# B&R Automation Studio project 305841_E00002_0
Automation Studio 4.10.3.60 SP; technology packages: mapp 5.16.1, mappCockpit 5.16.0, mappControl 5.16.0, mappMotion 5.16.2, mappSafety 5.16.0, mappView 5.16.1

## Configuration EchCm_AM

CPU X20CP3586, AutomationRuntime B4.92, Build 6.3.0, Safety 0.0, Vc V4.72.5

### Task classes (Cpu.sw)
```
Cyclic#2 (cycle 6400 us, tolerance 6400 us):
  ProdCycle <- PlcLogic.ProdCycle.prg
  Annunc <- PlcLogic.Annunc.prg
Cyclic#3 (cycle 12000 us, tolerance 12000 us):
  Pendant <- PlcLogic.Pendant.prg
  ProcInputs <- PlcLogic.ProcInputs.prg
  axSpinSM <- PlcLogic.axSpindle.axSpindleSM.prg
  axOutESM <- PlcLogic.axOutE.axOutESM.prg
  axInESM <- PlcLogic.axInE.axInESM.prg
  axZSM <- PlcLogic.axZ.axZSM.prg
  axHwSM <- PlcLogic.axHandwheel.axHwSM.prg
  axCfVfdSM <- PlcLogic.axCfVfd.axCfVfdSM.prg
Cyclic#4 (cycle 48000 us, tolerance 48000 us):
  AxEnable <- PlcLogic.AxEnable.prg
  CuttingFlu <- PlcLogic.CuttingFluidVFD.prg
  OmSafeDev <- PlcLogic.OmSafeDev.prg
  CrCamTbl <- PlcLogic.CutProfile.CutProfileCam.prg
  CutProfile <- PlcLogic.CutProfile.PartCfgCalcs.prg
DataObjects: McAcpSys
NcDataObjects: axSpindleP <- PlcLogic.axSpindle.axSpindleParamTable.dob, axOutEPara <- PlcLogic.axOutE.axOutEParamTable.dob, axInEParam <- PlcLogic.axInE.axInEParamTable.dob, axZParamTa <- PlcLogic.axZ.axZParamTable.dob, Cam1P <- PlcLogic.axInE.Cam1P.dob, Cam1P_Fp <- PlcLogic.axInE.Cam1P_Fp.dob, Cam2P <- PlcLogic.axInE.Cam2P.dob, Cam2P_Fp <- PlcLogic.axInE.Cam2P_Fp.dob, Cam3P <- PlcLogic.axInE.Cam3P.dob, Cam3P_Fp <- PlcLogic.axInE.Cam3P_Fp.dob, Cam4P <- PlcLogic.axInE.Cam4P.dob, Cam4P_Fp <- PlcLogic.axInE.Cam4P_Fp.dob, Cam5P <- PlcLogic.axInE.Cam5P.dob, Cam5P_Fp <- PlcLogic.axInE.Cam5P_Fp.dob, Cam6P <- PlcLogic.axInE.Cam6P.dob, Cam6P_Fp <- PlcLogic.axInE.Cam6P_Fp.dob, McDriveLog
Binaries: udbdef, mvLoader, arflatprv, TCData, FWRules, arcoal, arsvcreg, McAcpSim, McProfGen, McAcpDrv, mCoWebSc, TCLang, OpcUaSrv, DataObject, Settings, iomap, asfw, axCfgZ, Role, ashwac, sysconf, arconfig, ashwd, Config, axCfgInE, axCfgSpin, asiol1, axCfgOutE, Anonymous, User, cockpit1, TC, vAxHwCfg, vAxHw, axCfgCfPmp, CamFeature, camlist1, mappConfig, angleLu, depthLu, vAxHwLin, vAxHwRot, wgRecipe, cmRecipe, HwLinCfg, Config_5, HwRotCfg, Config_3
Libraries: sys_lib, runtime, brsystem, GAProcIO, standard, McBase, SfDomain, MpAxis, McAxis, MpBase, MpRecipe, McAcpAx, GAMpMotion, McPureVAx, astime, AsBrStr, GAConvert, MpAlarmX, AsBrMath, GAMath, CoTrace, AsZip, FileIO, McDS402Ax, MTLookUp, astcp, asieccon, asiodiag, asepl, SfDomDrv, asusb, SfDomVis, aruser, arssl, powerlnk, MpSfDomMgr, dataobj, asioacc, GAMotor, MTFilter, MTBasics, MTTypes
```

### Hardware
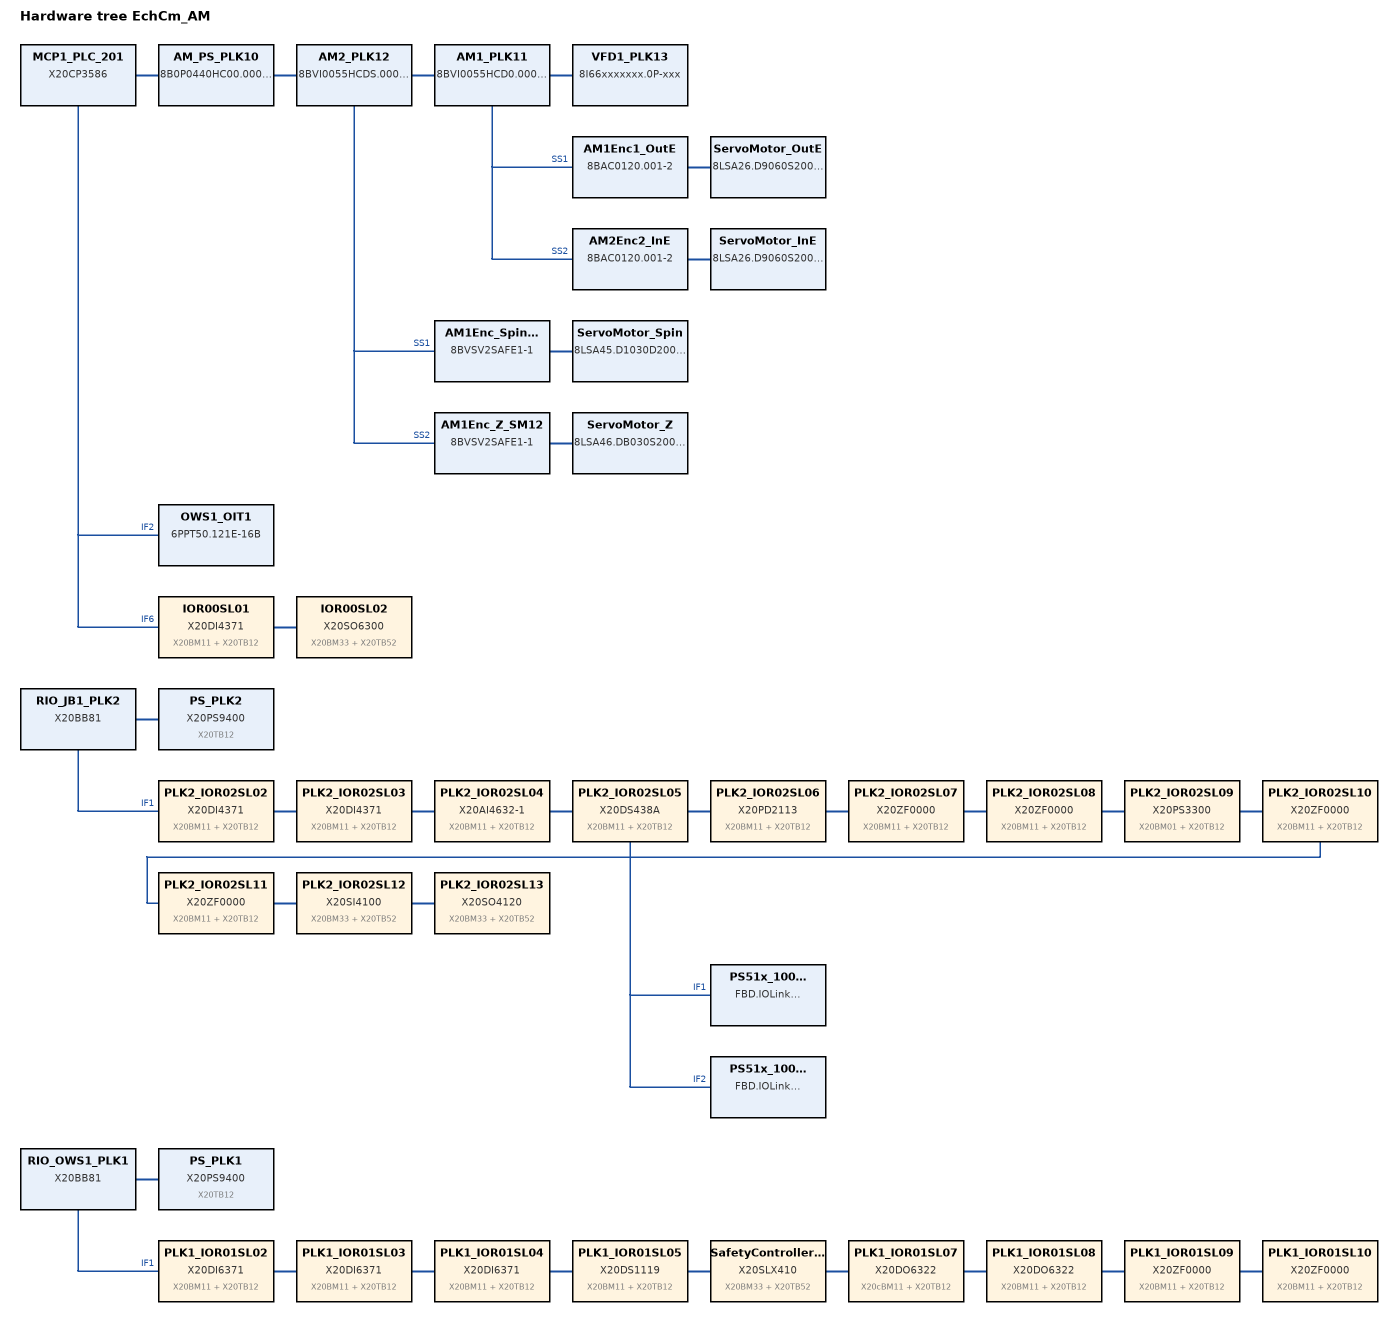
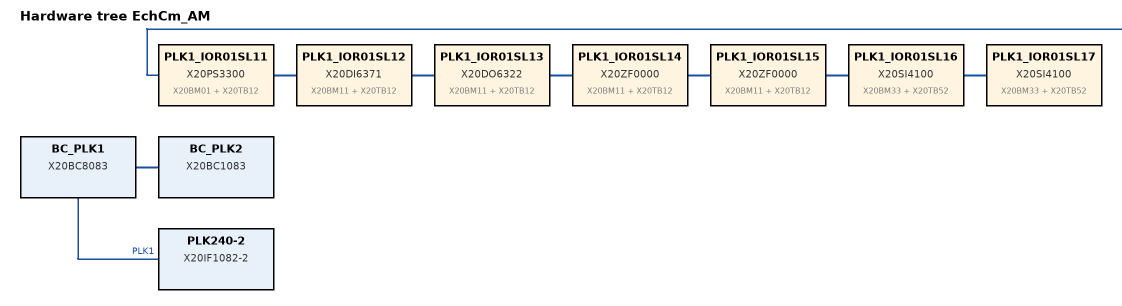
```
AM1Enc1_OutE : 8BAC0120.001-2 v2.2.0.0  [SS -> AM1_PLK11.SS1]
  PlugInType = Encoder
  McAcoposTypeID = AcoposMultiPlugInConfig
AM1Enc_Spin_SM11 : 8BVSV2SAFE1-1 v2.2.0.0  [SS -> AM2_PLK12.SS1]
  SafeModuleID = 11
  PlugInType = Encoder
  McAcoposTypeID = AcoposMultiPlugInConfig
AM1Enc_Z_SM12 : 8BVSV2SAFE1-1 v2.2.0.0  [SS -> AM2_PLK12.SS2]
  SafeModuleID = 12
  PlugInType = Encoder
  McAcoposTypeID = AcoposMultiPlugInConfig
AM1_PLK11 : 8BVI0055HCD0.000-1 v2.3.0.1  [PLK1 -> AM2_PLK12.PLK2 (NodeNumber=11) [Cable Type=PowerlinkCable, Length=10, Version=1.0.0.3]; PLK2 -> VFD1_PLK13.PLK1 (NodeNumber=11) [Cable Type=PowerlinkCable, Length=10, Version=1.0.0.3]; MT2 -> ServoMotor_InE.MT]
  DriveConfiguration/Module:
    McAcoposTypeID = AcoposP3SConfig
    ActivateACOPOSSimulationOnPLC = 0
  DriveConfiguration/Module/PowerSupply:
    PowerSupplyModuleReference = AM_PS
  DriveConfiguration/Channel[1]/RealAxis:
    AxisReference = gAxOutE
    MechanicalElementsIsInvisible = 0
  DriveConfiguration/Channel[1]/RealAxis/MechanicalElements/Gearbox:
    InputIsReadOnly = 0
    Input = 25
    OutputIsReadOnly = 0
    Output = 1
  DriveConfiguration/Channel[1]/RealAxis/MechanicalElements/RotaryToLinearTransformation:
    ReferenceDistanceIsReadOnly = 0
    ReferenceDistance = 360.0
  DriveConfiguration/Channel[1]/RealAxis/Controller:
    ModeIsReadOnly = 0
    Mode = PositionController
  DriveConfiguration/Channel[1]/RealAxis/Controller/Mode/Position:
    ProportionalGain = 462
    IntegrationTime = 0.1
    PredictionTime = 0.0004
    TotalDelayTime = 0.0004
  DriveConfiguration/Channel[1]/RealAxis/Controller/Mode/Speed:
    ProportionalGainIsReadOnly = 0
    ProportionalGain = 0.35
    IntegrationTimeIsReadOnly = 0
    IntegrationTime = 0.0
    FilterTimeIsReadOnly = 0
    FilterTime = 0.0
  DriveConfiguration/Channel[1]/RealAxis/Controller/Mode/LoopFilters:
    LoopFilterXIsReadOnly = 0
    LoopFilter1 = NotUsed
    LoopFilter2 = NotUsed
    LoopFilter3 = NotUsed
  DriveConfiguration/Channel[1]/RealAxis/Homing:
    ModeIsReadOnly = 0
    Mode = RestorePosition
    RestorePositionVariable = ::gr_AxOutERestorePos
  DriveConfiguration/Channel[1]/RealAxis/StopReaction:
    QuickstopIsReadOnly = 0
    Quickstop = DecelerationLimit
    DriveErrorIsReadOnly = 0
    DriveError = DecelerationLimit
  DriveConfiguration/Channel[1]/RealAxis/MovementErrorLimits:
    PositionError = 1.0
    VelocityErrorMonitoring = Automatic1
  DriveConfiguration/Channel[1]/RealAxis:
    JerkFilterIsReadOnly = 0
    JerkFilter = NotUsed
  DriveConfiguration/Channel[1]/RealAxis/DigitalInputs/HomingSwitch:
    SourceIsReadOnly = 0
    Source = NotUsed
    Level = High
  DriveConfiguration/Channel[1]/RealAxis/DigitalInputs/PositiveLimitSwitch:
    SourceIsReadOnly = 0
    Source = NotUsed
    Level = High
  DriveConfiguration/Channel[1]/RealAxis/DigitalInputs/NegativeLimitSwitch:
    SourceIsReadOnly = 0
    Source = NotUsed
    Level = High
  DriveConfiguration/Channel[1]/RealAxis/DigitalInputs/Trigger1:
    Source = X2Trigger1
    Level = High
  DriveConfiguration/Channel[1]/RealAxis/DigitalInputs/Trigger2:
    Source = X2Trigger2
    Level = High
  DriveConfiguration/Channel[1]/RealAxis/DigitalInputs/Quickstop:
    Input = NotUsed
  DriveConfiguration/Channel[1]/RealAxis/Simulation:
    SimulationModeOnPLC = SetValueGeneration
    SimulationModeOnACOPOS = NotUsed
  DriveConfiguration/Channel[1]:
    ExternalEncoderAxis = NotUsed
  DriveConfiguration/Channel[2]/RealAxis:
    AxisReference = gAxInE
    MechanicalElementsIsInvisible = 0
  DriveConfiguration/Channel[2]/RealAxis/MechanicalElements/Gearbox:
    InputIsReadOnly = 0
    Input = 25
    OutputIsReadOnly = 0
    Output = 1
  DriveConfiguration/Channel[2]/RealAxis/MechanicalElements/RotaryToLinearTransformation:
    ReferenceDistanceIsReadOnly = 0
    ReferenceDistance = 360.0
  DriveConfiguration/Channel[2]/RealAxis/Controller:
    ModeIsReadOnly = 0
    Mode = PositionController
  DriveConfiguration/Channel[2]/RealAxis/Controller/Mode/Position:
    ProportionalGain = 451.5
    IntegrationTime = 0.1
    PredictionTime = 0.0004
    TotalDelayTime = 0.0004
  DriveConfiguration/Channel[2]/RealAxis/Controller/Mode/Speed:
    ProportionalGainIsReadOnly = 0
    ProportionalGain = 0.325
    IntegrationTimeIsReadOnly = 0
    IntegrationTime = 0.0
    FilterTimeIsReadOnly = 0
    FilterTime = 0.0
  DriveConfiguration/Channel[2]/RealAxis/Controller/Mode/LoopFilters:
    LoopFilterXIsReadOnly = 0
    LoopFilter1 = NotUsed
    LoopFilter2 = NotUsed
    LoopFilter3 = NotUsed
  DriveConfiguration/Channel[2]/RealAxis/Homing:
    ModeIsReadOnly = 0
    Mode = RestorePosition
    RestorePositionVariable = ::gr_AxInERestorePos
  DriveConfiguration/Channel[2]/RealAxis/StopReaction:
    QuickstopIsReadOnly = 0
    Quickstop = DecelerationLimit
    DriveErrorIsReadOnly = 0
    DriveError = DecelerationLimit
  DriveConfiguration/Channel[2]/RealAxis/MovementErrorLimits:
    PositionError = 0.9
    VelocityErrorMonitoring = Automatic1
  DriveConfiguration/Channel[2]/RealAxis:
    JerkFilterIsReadOnly = 0
    JerkFilter = NotUsed
  DriveConfiguration/Channel[2]/RealAxis/DigitalInputs/HomingSwitch:
    SourceIsReadOnly = 0
    Source = NotUsed
    Level = High
  DriveConfiguration/Channel[2]/RealAxis/DigitalInputs/PositiveLimitSwitch:
    SourceIsReadOnly = 0
    Source = NotUsed
    Level = Low
  DriveConfiguration/Channel[2]/RealAxis/DigitalInputs/NegativeLimitSwitch:
    SourceIsReadOnly = 0
    Source = NotUsed
    Level = Low
  DriveConfiguration/Channel[2]/RealAxis/DigitalInputs/Trigger1:
    Source = X2Trigger1
    Level = High
  DriveConfiguration/Channel[2]/RealAxis/DigitalInputs/Trigger2:
    Source = X2Trigger2
    Level = High
  DriveConfiguration/Channel[2]/RealAxis/DigitalInputs/Quickstop:
    Input = NotUsed
  DriveConfiguration/Channel[2]/RealAxis/Simulation:
    SimulationModeOnPLC = SetValueGeneration
    SimulationModeOnACOPOS = NotUsed
  DriveConfiguration/Channel[2]/RealAxis/AxisFeatures:
    FeatureRef[1] = 
  DriveConfiguration/Channel[2]:
    ExternalEncoderAxis = NotUsed
  DriveConfiguration/Channel[2]/ChannelFeatures:
    FeatureRef[1] = Feature_CamList
AM2Enc2_InE : 8BAC0120.001-2 v2.2.0.0  [SS -> AM1_PLK11.SS2]
  PlugInType = Encoder
  McAcoposTypeID = AcoposMultiPlugInConfig
AM2_PLK12 : 8BVI0055HCDS.000-1 v2.3.0.1  [PLK1 -> AM_PS_PLK10.PLK2 (NodeNumber=12) [Cable Type=PowerlinkCable, Length=10, Version=1.0.0.3]; PLK2 -> AM1_PLK11.PLK1 (NodeNumber=12) [Cable Type=PowerlinkCable, Length=10, Version=1.0.0.3]; MT2 -> ServoMotor_Z.MT]
  DriveConfiguration/Module:
    McAcoposTypeID = AcoposMultiDConfig
    ActivateACOPOSSimulationOnPLC = 0
  DriveConfiguration/Module/PowerSupply:
    PowerSupplyModuleReference = AM_PS
  DriveConfiguration/Channel[1]/RealAxis:
    AxisReference = gAxSpin
    MechanicalElementsIsInvisible = 0
  DriveConfiguration/Channel[1]/RealAxis/MechanicalElements/Gearbox:
    InputIsReadOnly = 0
    Input = 1
    OutputIsReadOnly = 0
    Output = 1
  DriveConfiguration/Channel[1]/RealAxis/MechanicalElements/RotaryToLinearTransformation:
    ReferenceDistanceIsReadOnly = 0
    ReferenceDistance = 1
  DriveConfiguration/Channel[1]/RealAxis/Controller:
    ModeIsReadOnly = 0
    Mode = PositionControllerWithTorqueFeedForward
  DriveConfiguration/Channel[1]/RealAxis/Controller/Mode/Position:
    ProportionalGainIsReadOnly = 0
    ProportionalGain = 200
    IntegrationTimeIsReadOnly = 0
    IntegrationTime = 0.0
    TotalDelayTime = 0.0004
  DriveConfiguration/Channel[1]/RealAxis/Controller/Mode/Speed:
    ProportionalGainIsReadOnly = 0
    ProportionalGain = 0.25
    IntegrationTimeIsReadOnly = 0
    IntegrationTime = 0
    FilterTimeIsReadOnly = 0
    FilterTime = 0
  DriveConfiguration/Channel[1]/RealAxis/Controller/Mode:
    FeedForwardIsReadOnly = 0
    FeedForward = Standard
  DriveConfiguration/Channel[1]/RealAxis/Controller/Mode/FeedForward:
    TorqueLoad = 0.0
    TorquePositive = 0.3405416
    TorqueNegative = 0.3405416
    SpeedTorqueFactor = 0.00008983436
    Inertia = 0.00009823628
    AccelerationFilterTime = 0.0
  DriveConfiguration/Channel[1]/RealAxis/Controller/Mode/LoopFilters:
    LoopFilterXIsReadOnly = 0
    LoopFilter1 = NotUsed
    LoopFilter2 = NotUsed
    LoopFilter3 = NotUsed
  DriveConfiguration/Channel[1]/RealAxis/Homing:
    ModeIsReadOnly = 0
    Mode = RestorePosition
    RestorePositionVariable = ::gr_AxSpinRestorePos
  DriveConfiguration/Channel[1]/RealAxis/StopReaction:
    QuickstopIsReadOnly = 0
    Quickstop = DecelerationLimit
    DriveErrorIsReadOnly = 0
    DriveError = DecelerationLimit
  DriveConfiguration/Channel[1]/RealAxis/MovementErrorLimits:
    PositionError = 2
    VelocityErrorMonitoring = Automatic1
  DriveConfiguration/Channel[1]/RealAxis:
    JerkFilterIsReadOnly = 0
    JerkFilter = NotUsed
  DriveConfiguration/Channel[1]/RealAxis/DigitalInputs/HomingSwitch:
    SourceIsReadOnly = 0
    Source = NotUsed
    Level = High
  DriveConfiguration/Channel[1]/RealAxis/DigitalInputs/PositiveLimitSwitch:
    SourceIsReadOnly = 0
    Source = NotUsed
    Level = High
  DriveConfiguration/Channel[1]/RealAxis/DigitalInputs/NegativeLimitSwitch:
    SourceIsReadOnly = 0
    Source = NotUsed
    Level = High
  DriveConfiguration/Channel[1]/RealAxis/DigitalInputs/Trigger1:
    Source = X2Trigger1
    Level = High
  DriveConfiguration/Channel[1]/RealAxis/DigitalInputs/Trigger2:
    Source = X2Trigger2
    Level = High
  DriveConfiguration/Channel[1]/RealAxis/DigitalInputs/Quickstop:
    Input = NotUsed
  DriveConfiguration/Channel[1]/RealAxis/Simulation:
    SimulationModeOnPLC = SetValueGeneration
    SimulationModeOnACOPOS = NotUsed
  DriveConfiguration/Channel[1]:
    ExternalEncoderAxis = NotUsed
  DriveConfiguration/Channel[2]/RealAxis:
    AxisReference = gAxZ
    MechanicalElementsIsInvisible = 0
  DriveConfiguration/Channel[2]/RealAxis/MechanicalElements/Gearbox:
    InputIsReadOnly = 0
    Input = 1
    OutputIsReadOnly = 0
    Output = 1
  DriveConfiguration/Channel[2]/RealAxis/MechanicalElements/RotaryToLinearTransformation:
    ReferenceDistanceIsReadOnly = 0
    ReferenceDistance = 5.00
  DriveConfiguration/Channel[2]/RealAxis/Controller:
    ModeIsReadOnly = 0
    Mode = PositionController
  DriveConfiguration/Channel[2]/RealAxis/Controller/Mode/Position:
    ProportionalGain = 551
    IntegrationTime = 0.0
    PredictionTime = 0.0004
    TotalDelayTime = 0.0004
  DriveConfiguration/Channel[2]/RealAxis/Controller/Mode/Speed:
    ProportionalGainIsReadOnly = 0
    ProportionalGain = 1.0
    IntegrationTimeIsReadOnly = 0
    IntegrationTime = 0.0
    FilterTimeIsReadOnly = 0
    FilterTime = 0.0
  DriveConfiguration/Channel[2]/RealAxis/Controller/Mode/LoopFilters:
    LoopFilterXIsReadOnly = 0
    LoopFilter1 = NotUsed
    LoopFilter2 = NotUsed
    LoopFilter3 = NotUsed
  DriveConfiguration/Channel[2]/RealAxis/Homing:
    ModeIsReadOnly = 0
    Mode = RestorePosition
    RestorePositionVariable = ::gr_AxZRestorePos
  DriveConfiguration/Channel[2]/RealAxis/StopReaction:
    QuickstopIsReadOnly = 0
    Quickstop = DecelerationLimit
    DriveErrorIsReadOnly = 0
    DriveError = DecelerationLimit
  DriveConfiguration/Channel[2]/RealAxis/MovementErrorLimits:
    PositionError = 1.0
    VelocityErrorMonitoring = Automatic1
  DriveConfiguration/Channel[2]/RealAxis:
    JerkFilterIsReadOnly = 0
    JerkFilter = NotUsed
  DriveConfiguration/Channel[2]/RealAxis/DigitalInputs/HomingSwitch:
    SourceIsReadOnly = 0
    Source = NotUsed
    Level = High
  DriveConfiguration/Channel[2]/RealAxis/DigitalInputs/PositiveLimitSwitch:
    SourceIsReadOnly = 0
    Source = X2Trigger1
    Level = Low
  DriveConfiguration/Channel[2]/RealAxis/DigitalInputs/NegativeLimitSwitch:
    SourceIsReadOnly = 0
    Source = X2Trigger2
    Level = Low
  DriveConfiguration/Channel[2]/RealAxis/DigitalInputs/Trigger1:
    Source = X2Trigger1
    Level = High
  DriveConfiguration/Channel[2]/RealAxis/DigitalInputs/Trigger2:
    Source = X2Trigger2
    Level = High
  DriveConfiguration/Channel[2]/RealAxis/DigitalInputs/Quickstop:
    Input = NotUsed
  DriveConfiguration/Channel[2]/RealAxis/Simulation:
    SimulationModeOnPLC = SetValueGeneration
    SimulationModeOnACOPOS = NotUsed
  DriveConfiguration/Channel[2]/RealAxis/AxisFeatures:
    FeatureRef[1] = 
  DriveConfiguration/Channel[2]:
    ExternalEncoderAxis = NotUsed
AM_PS_PLK10 : 8B0P0440HC00.000-1 v2.3.0.1  [PLK1 -> MCP1_PLC_201.IF3 (NodeNumber=10) [Cable Type=PowerlinkCable, Length=10, Version=1.0.0.3]; PLK2 -> AM2_PLK12.PLK1 (NodeNumber=10) [Cable Type=PowerlinkCable, Length=10, Version=1.0.0.3]]
  DriveConfiguration/Module:
    McAcoposTypeID = AcoposMultiPSMpConfig
    ActivateACOPOSSimulationOnPLC = 0
  DriveConfiguration/Channel[1]/PowerSection:
    AxisReference = AM_PS
BC_PLK1 : X20BC8083 v2.14.0.0  [PLK1 -> PLK240-2.PLK2 (NodeNumber=1) [Cable Type=PowerlinkCable, Length=10, Version=1.0.0.3]; PLK2 -> BC_PLK2.PLK1 (NodeNumber=1) [Cable Type=PowerlinkCable, Length=10, Version=1.0.0.3]; SL -> RIO_OWS1_PLK1.SL1]
BC_PLK2 : X20BC1083 v2.14.0.0  [PLK1 -> BC_PLK1.PLK2 (NodeNumber=2) [Cable Type=PowerlinkCable, Length=10, Version=1.0.0.3]; SL -> RIO_JB1_PLK2.SL1]
IOR00SL01 : X20DI4371 v1.2.0.0  [SS1 -> X20TB12.SS; SL -> X20BM11.SL1]
IOR00SL02 : X20SO6300 v2.3.0.0  [SS1 -> X20TB52d.SS; SL -> X20BM33d.SL1]
  DigitalOutput01 = viaSafeLOGIC
  DigitalOutput02 = viaSafeLOGIC
  DigitalOutput03 = viaSafeLOGIC
  DigitalOutput04 = viaSafeLOGIC
  DigitalOutput05 = viaSafeLOGIC
  DigitalOutput06 = viaSafeLOGIC
MCP1_PLC_201 : X20CP3586 v1.10.0.0
  Connector IF2:
    ActivateDevice = 1
    HostName = plc_mcp1
    Mode = Manual
    InternetAddress = 10.10.2.240
    SubnetMask = 255.255.255.0
  Connector IF3:
    EplHostName = PLC_MCP1_PLK1
    CycleTime = 800
  Connector IF6:
    CycleTime = 800
  ConfigurationID = 305841_E00002_Rev0_PLC_Main
  ConfigVersion = 0.0.0
  UserPartitionSize = 20
  AutomaticTransferOfUserfiles = on
  PermanentPvSize = 9216
  VolatileGlobalPvSize = 69630
  TimerDeviceType = EPLX2X
  TimerDevice = MCP1_PLC_201.IF3
  TaskClassIdleTime = 800
  CyclicTaskClassCount = 6
  Cyclic1Duration = 800
  Cyclic1Tolerance = 800
  Cyclic2Duration = 6400
  Cyclic2Tolerance = 6400
  Cyclic3Duration = 12000
  Cyclic3Tolerance = 12000
  Cyclic4Duration = 48000
  Cyclic4Tolerance = 48000
  Cyclic5Duration = 96000
  Cyclic5Tolerance = 9600000
  Cyclic6Duration = 480000
  Cyclic6Tolerance = 480000
  Cyclic8Duration = 9600
  FileDevice1
  FileDeviceName1 = UserPartitionRoot
  FileDevicePath1 = F:\
  FileDevice2
  FileDeviceName2 = Recipes
  FileDevicePath2 = F:\config\recipes\
  FileDevice3
  FileDeviceName3 = IOConfig
  FileDevicePath3 = F:\config\io\
  EthernetHostName = mcp1_plc201
  FtpUser1
  FtpUsername1 = ftpuser
  FtpUserPassword1 = wzi3iB5UNI3uCms7ZCmB0Woh2QaOICjzuPm+LM5DkNg=
  FtpUserSalt1 = UFkRbDjT
  FTPAccessRight1 = 0
  ActivateOpcUa = 1
  OpcUaPort = 4841
  OpcUaInformationModels_PV_Version = 1
OWS1_OIT1 : 6PPT50.121E-16B v1.3.8.0  [ETH1 -> MCP1_PLC_201.IF2 [Cable Type=PowerlinkCable, Length=10, Version=1.0.0.3]]
  Terminal = true
  Mode = Manual
  InternetAddress = 10.10.2.20
  Subnetmask = 255.255.255.0
  Hostname = ows1_oit1
  PasswordVNC = 
  PasswordCIFS = 
  PasswordService = 
PLK1_IOR01SL02 : X20DI6371 v1.2.0.0  [SS1 -> X20TB12n.SS; SL -> X20BM11l.SL1]
  InputFilter = 250
PLK1_IOR01SL03 : X20DI6371 v1.2.0.0  [SS1 -> X20TB12c.SS; SL -> X20BM11c.SL1]
  InputFilter = 250
PLK1_IOR01SL04 : X20DI6371 v1.2.0.0  [SS1 -> X20TB12ab.SS; SL -> X20BM11x.SL1]
  InputFilter = 250
PLK1_IOR01SL05 : X20DS1119 v1.5.0.0  [SS1 -> X20TB12e.SS; SL -> X20BM11e.SL1]
  PSInfo = on
  SDCInfo = on
  NetworkInfo = 8Bit
  Function03 = AB
PLK1_IOR01SL07 : X20DO6322 v1.3.0.0  [SS1 -> X20TB12p.SS; SL -> X20cBM11a.SL1]
PLK1_IOR01SL08 : X20DO6322 v1.3.0.0  [SS1 -> X20TB12h.SS; SL -> X20BM11h.SL1]
PLK1_IOR01SL09 : X20ZF0000 v1.1.0.0 (Disabled=true)  [SS1 -> X20TB12o.SS; SL -> X20BM11n.SL1]
PLK1_IOR01SL10 : X20ZF0000 v1.1.0.0 (Disabled=true)  [SS1 -> X20TB12i.SS; SL -> X20BM11m.SL1]
PLK1_IOR01SL11 : X20PS3300 v1.4.0.0  [SS1 -> X20TB12z.SS; SL -> X20BM01.SL1]
  PowerInfo = on
PLK1_IOR01SL12 : X20DI6371 v1.2.0.0  [SS1 -> X20TB12d.SS; SL -> X20BM11d.SL1]
PLK1_IOR01SL13 : X20DO6322 v1.3.0.0  [SS1 -> X20TB12b.SS; SL -> X20BM11b.SL1]
  Supervision = off
PLK1_IOR01SL14 : X20ZF0000 v1.1.0.0 (Disabled=true)  [SS1 -> X20TB12f.SS; SL -> X20BM11f.SL1]
PLK1_IOR01SL15 : X20ZF0000 v1.1.0.0 (Disabled=true)  [SS1 -> X20TB12q.SS; SL -> X20BM11o.SL1]
PLK1_IOR01SL16 : X20SI4100 v2.4.0.0  [SS1 -> X20TB52b.SS; SL -> X20BM33b.SL1]
  SafeModuleID = 116
PLK1_IOR01SL17 : X20SI4100 v2.4.0.0  [SS1 -> X20TB52a.SS; SL -> X20BM33a.SL1]
  SafeModuleID = 117
PLK240-2 : X20IF1082-2 v1.14.0.0  [PLK2 -> BC_PLK1.PLK1 [Cable Type=PowerlinkCable, Length=10, Version=1.0.0.3]; SS -> MCP1_PLC_201.SS1]
  Connector IF1:
    EplHostName = PLC_MCP1_PLK2
    CycleTime = 800
    NodeDefinition = Software
    EplNatSubnet = 192.168.102.0
PLK2_IOR02SL02 : X20DI4371 v1.2.0.0  [SS1 -> X20TB12s.SS; SL -> X20BM11p.SL1]
PLK2_IOR02SL03 : X20DI4371 v1.2.0.0  [SS1 -> X20TB12t.SS; SL -> X20BM11q.SL1]
PLK2_IOR02SL04 : X20AI4632-1 v1.2.0.0  [SS1 -> X20TB12u.SS; SL -> X20BM11r.SL1]
  ChannelType01 = 0 to 22mA
  ChannelType02 = 0 to 22mA
  Channel03enable = off
  Channel04enable = off
PLK2_IOR02SL05 : X20DS438A v2.4.0.0  [SS1 -> X20TB12aa.SS; SL -> X20BM11w.SL1]
  DtmRef = FBD.BRIOLinkModuleDTM.DTMCore.X20DS438A
  DtmId = 7db43003-0ff5-4bbd-8923-86eacecae911
  CommDtmId = ab9d1316-8c35-4493-ab34-f7b1b8ca9169
  RequiresDTMBuild = true
  ConfigFile = Communication.dtm
  ConfigModule = asiol1
  OperatingMode01 = Operate
  PDI_Enable01 = variousTypes
  PDI_DataType01_1 = UINT
  OperatingMode02 = Operate
  PDI_Enable02 = variousTypes
  PDI_DataType02_1 = UINT
PLK2_IOR02SL06 : X20PD2113 v1.2.0.0  [SS1 -> X20TB12g.SS; SL -> X20BM11g.SL1]
PLK2_IOR02SL07 : X20ZF0000 v1.1.0.0 (Disabled=true)  [SS1 -> X20TB12x.SS; SL -> X20BM11t.SL1]
PLK2_IOR02SL08 : X20ZF0000 v1.1.0.0 (Disabled=true)  [SS1 -> X20TB12w.SS; SL -> X20BM11v.SL1]
PLK2_IOR02SL09 : X20PS3300 v1.4.0.0 (Disabled=true)  [SS1 -> X20TB12ac.SS; SL -> X20BM01a.SL1]
  PowerInfo = on
PLK2_IOR02SL10 : X20ZF0000 v1.1.0.0 (Disabled=true)  [SS1 -> X20TB12y.SS; SL -> X20BM11u.SL1]
PLK2_IOR02SL11 : X20ZF0000 v1.1.0.0 (Disabled=true)  [SS1 -> X20TB12v.SS; SL -> X20BM11s.SL1]
PLK2_IOR02SL12 : X20SI4100 v2.4.0.0  [SS1 -> X20TB52c.SS; SL -> X20BM33c.SL1]
  SafeModuleID = 212
PLK2_IOR02SL13 : X20SO4120 v2.3.0.0  [SS1 -> X20TB52e.SS; SL -> X20BM33e.SL1]
  PLCopenInfo = on
  SafeModuleID = 213
  DigitalOutput01 = viaSafeLOGIC
  DigitalOutput02 = viaSafeLOGIC
  DigitalOutput03 = viaSafeLOGIC
  DigitalOutput04 = viaSafeLOGIC
PS51x_100_LI2UPN8_IODD1_1 : FBD.IOLink.GenericDeviceDTM.DTMCore.PS51x-100-LI2UPN8 IODD1.1 v2.9 (OrderNumber=PS51x-100-LI2UPN8 IODD1.1)  [IO-Link1 -> PLK2_IOR02SL05.IF1]
  DtmId = 9f03f336-de2c-4174-a814-ce0739b6707c
PS51x_100_LI2UPN8_IODD1_1a : FBD.IOLink.GenericDeviceDTM.DTMCore.PS51x-100-LI2UPN8 IODD1.1 v2.9 (OrderNumber=PS51x-100-LI2UPN8 IODD1.1)  [IO-Link1 -> PLK2_IOR02SL05.IF2]
  DtmId = 948ae1a5-f93f-40dc-8e06-a46fa964d649
PS_PLK1 : X20PS9400 v1.8.0.0  [SS1 -> X20TB12m.SS; PS -> RIO_OWS1_PLK1.PS1]
  PowerInfo = on
PS_PLK2 : X20PS9400 v1.8.0.0  [SS1 -> X20TB12r.SS; PS -> RIO_JB1_PLK2.PS1]
RIO_JB1_PLK2 : X20BB81 v1.1.0.0
  Connector IF1:
    CycleTime = 800
RIO_OWS1_PLK1 : X20BB81 v1.1.0.0
  Connector IF1:
    CycleTime = 800
SafetyController_R01SL06 : X20SLX410 v2.4.1.1  [SS1 -> X20TB52.SS; SL -> X20BM33.SL1]
  UnsafeOutputBOOLs = 24
  UnsafeInputBOOLs = 24
  UnsafeInputUINTs = 4
ServoMotor_InE : 8LSA26.D9060S200-3 v2.2.0.1  [EC -> AM2Enc2_InE.EC; MT -> AM1_PLK11.MT2]
  M1/MotorParameters:
    MOTOR_AMB_TEMP_RATED = 40
ServoMotor_OutE : 8LSA26.D9060S200-3 v2.2.0.1  [EC -> AM1Enc1_OutE.EC; MT -> AM1_PLK11.MT1]
  M1/MotorParameters:
    MOTOR_AMB_TEMP_RATED = 40
ServoMotor_Spin : 8LSA45.D1030D200-0 v1.0.5.35  [EC -> AM1Enc_Spin_SM11.EC; MT -> AM2_PLK12.MT1]
ServoMotor_Z : 8LSA46.DB030S200-3 v2.2.0.1  [EC -> AM1Enc_Z_SM12.EC; MT -> AM2_PLK12.MT2]
  M1/MotorParameters:
    MOTOR_AMB_TEMP_RATED = 40
VFD1_PLK13 : 8I66xxxxxxx.0P-xxx v2.5.1.0  [PLK1 -> AM1_PLK11.PLK2 (NodeNumber=13) [Cable Type=PowerlinkCable, Length=10, Version=1.0.0.3]]
  Supervision = off
  PlkDiagnosisAdd = on
  FunctionModel = MotionConfig
  McTypeID = McAcoposInverterP66P
  AxisReference = gAxCfPmp
  InputIsReadOnly = 0
  Input = 1
  OutputIsReadOnly = 0
  Output = 1
  ReferenceDistanceIsReadOnly = 0
  ReferenceDistance = 1
  UnitOfSetpoint = Rpm
  IOM_AIDP1 = HMIS
  IOM_AIDP2 = LFT
  IOM_AIDP3 = ETAD_u
  Mode_LI3 = Safety
  Sel_NameplateMask = 8Ix6T401100_IEC
  Cfg_NSP = 1175
  Cfg_FRS = 600
  Cfg_UNS = 480
  Cfg_COS = 73
X20BM01 : X20BM01 v2.1.0.0  [X2X1 -> X20BM11m.X2X2]
X20BM01a : X20BM01 v2.1.0.0 (Disabled=true)  [X2X1 -> X20BM11v.X2X2]
X20BM11 : X20BM11 v1.1.0.0  [X2X1 -> MCP1_PLC_201.IF6]
X20BM11b : X20BM11 v1.1.0.0  [X2X1 -> X20BM11d.X2X2]
X20BM11c : X20BM11 v1.1.0.0  [X2X1 -> X20BM11l.X2X2]
X20BM11d : X20BM11 v1.1.0.0  [X2X1 -> X20BM01.X2X2]
X20BM11e : X20BM11 v1.1.0.0  [X2X1 -> X20BM11x.X2X2]
X20BM11f : X20BM11 v1.1.0.0 (Disabled=true)  [X2X1 -> X20BM11b.X2X2]
X20BM11g : X20BM11 v1.1.0.0  [X2X1 -> X20BM11w.X2X2]
X20BM11h : X20BM11 v1.1.0.0  [X2X1 -> X20cBM11a.X2X2]
X20BM11l : X20BM11 v1.1.0.0  [X2X1 -> RIO_OWS1_PLK1.IF1]
X20BM11m : X20BM11 v1.1.0.0 (Disabled=true)  [X2X1 -> X20BM11n.X2X2]
X20BM11n : X20BM11 v1.1.0.0 (Disabled=true)  [X2X1 -> X20BM11h.X2X2]
X20BM11o : X20BM11 v1.1.0.0 (Disabled=true)  [X2X1 -> X20BM11f.X2X2]
X20BM11p : X20BM11 v1.1.0.0  [X2X1 -> RIO_JB1_PLK2.IF1]
X20BM11q : X20BM11 v1.1.0.0  [X2X1 -> X20BM11p.X2X2]
X20BM11r : X20BM11 v1.1.0.0  [X2X1 -> X20BM11q.X2X2]
X20BM11s : X20BM11 v1.1.0.0 (Disabled=true)  [X2X1 -> X20BM11u.X2X2]
X20BM11t : X20BM11 v1.1.0.0 (Disabled=true)  [X2X1 -> X20BM11g.X2X2]
X20BM11u : X20BM11 v1.1.0.0 (Disabled=true)  [X2X1 -> X20BM01a.X2X2]
X20BM11v : X20BM11 v1.1.0.0 (Disabled=true)  [X2X1 -> X20BM11t.X2X2]
X20BM11w : X20BM11 v1.1.0.0  [X2X1 -> X20BM11r.X2X2]
X20BM11x : X20BM11 v1.1.0.0  [X2X1 -> X20BM11c.X2X2]
X20BM33 : X20BM33 v1.0.0.6  [X2X1 -> X20BM11e.X2X2]
X20BM33a : X20BM33 v1.0.0.6  [X2X1 -> X20BM33b.X2X2]
X20BM33b : X20BM33 v1.0.0.6  [X2X1 -> X20BM11o.X2X2]
X20BM33c : X20BM33 v1.0.0.6  [X2X1 -> X20BM11s.X2X2]
X20BM33d : X20BM33 v1.0.0.6  [X2X1 -> X20BM11.X2X2]
X20BM33e : X20BM33 v1.0.0.6  [X2X1 -> X20BM33c.X2X2]
X20TB12 : X20TB12 v1.0.0.0
X20TB12aa : X20TB12 v1.0.0.0
X20TB12ab : X20TB12 v1.0.0.0
X20TB12ac : X20TB12 v1.0.0.0 (Disabled=true)
X20TB12b : X20TB12 v1.0.0.0
X20TB12c : X20TB12 v1.0.0.0
X20TB12d : X20TB12 v1.0.0.0
X20TB12e : X20TB12 v1.0.0.0
X20TB12f : X20TB12 v1.0.0.0 (Disabled=true)
X20TB12g : X20TB12 v1.0.0.0
X20TB12h : X20TB12 v1.0.0.0
X20TB12i : X20TB12 v1.0.0.0 (Disabled=true)
X20TB12m : X20TB12 v1.0.0.0
X20TB12n : X20TB12 v1.0.0.0
X20TB12o : X20TB12 v1.0.0.0 (Disabled=true)
X20TB12p : X20TB12 v1.0.0.0
X20TB12q : X20TB12 v1.0.0.0 (Disabled=true)
X20TB12r : X20TB12 v1.0.0.0
X20TB12s : X20TB12 v1.0.0.0
X20TB12t : X20TB12 v1.0.0.0
X20TB12u : X20TB12 v1.0.0.0
X20TB12v : X20TB12 v1.0.0.0 (Disabled=true)
X20TB12w : X20TB12 v1.0.0.0 (Disabled=true)
X20TB12x : X20TB12 v1.0.0.0 (Disabled=true)
X20TB12y : X20TB12 v1.0.0.0 (Disabled=true)
X20TB12z : X20TB12 v1.0.0.0
X20TB52 : X20TB52 v1.0.0.2
X20TB52a : X20TB52 v1.0.0.2
X20TB52b : X20TB52 v1.0.0.2
X20TB52c : X20TB52 v1.0.0.2
X20TB52d : X20TB52 v1.0.0.2
X20TB52e : X20TB52 v1.0.0.2
X20cBM11a : X20cBM11 v1.0.1.0  [X2X1 -> X20BM33.X2X2]
```

### Cpu.per - MCP1_PLC_201/Cpu.per
```iecst
VAR_CONFIG
	gr_AxSpindleRestorePos AT %M0; (* *)
	gr_AxOutERestorePos AT %M72; (* *)
	gr_AxInERestorePos AT %M144; (* *)
	gr_AxZRestorePos AT %M216; (* *)
	gr_AI_FT_CFFlow_Params AT %M288; (* *)
	gr_AI_LT_CFTankLevel_Params AT %M376; (* *)
	gr_AI_PT_CFFilterOutlet_Params AT %M464; (* *)
	gr_AI_PT_CFPumpOutlet_Params AT %M552; (* *)
	gr_AI_DP_CFFilter_Params AT %M640; (* *)
	gr_DI_JI_480VACOk_Params AT %M728; (* *)
	gr_DI_LSL_CFTank_Params AT %M760; (* *)
	gr_DI_ZS_CFTankLocator_Params AT %M792; (* *)
	gr_AxisPositionLimits AT %M824; (* *)
	gr_CfgCurrent AT %M968; (* *)
	gr_PartCurrent AT %M1172; (* *)
	gr_depthToAngleLu AT %M1288; (* *)
	gr_angleToDepthLu AT %M2500; (* *)
	gr_ProdModeStepTOs AT %MD3712; (*step Timeout time values *)
	gr_ProdModeStepMins AT %MD3876; (*step minimum time values *)
END_VAR
```

### axCfgInE.axis - MCP1_PLC_201/mappMotion/Eccentrics/axCfgInE.axis
```
Element gAxInE (Type=axis)
  BaseTypeIsReadOnly = 0
  BaseType = RotaryPeriodic
    MeasurementUnitIsReadOnly = 0
    MeasurementUnit = 17476
    MeasurementResolutionIsReadOnly = 0
    MeasurementResolution = 0.001
    CountDirectionIsReadOnly = 0
    CountDirection = Inverse
    PeriodSettings:
      Period = 360.0
  MovementLimitsIsReadOnly = 0
  MovementLimits = Internal
    Position:
      LowerLimitMin = -1.79769313486231E308
      UpperLimitMax = 1.79769313486231E308
      LowerLimit = -1000.0
      UpperLimit = 1000.0
    VelocityIsReadOnly = 0
    Velocity:
      VelocityMax = 3.4E38
      Velocity = 1600
    AccelerationIsReadOnly = 0
    Acceleration:
      AccelerationMax = 3.4E38
      Acceleration = 1600
    DecelerationIsReadOnly = 0
    Deceleration:
      DecelerationMax = 3.4E38
      Deceleration = 6000
  Alarms = MpAlarmX
```

### camlist1.camlist - MCP1_PLC_201/mappMotion/Eccentrics/camlist1.camlist
```
Element CamList_1 (Type=camlist)
  Row[1]:
    CamName = Cam1P
    CamID = 1
    Description
  Row[2]:
    CamName = Cam1P_Fp
    CamID = 2
    Description
  Row[3]:
    CamName = Cam2P
    CamID = 3
    Description
  Row[4]:
    CamName = Cam2P_Fp
    CamID = 4
    Description
  Row[5]:
    CamName = Cam3P
    CamID = 5
    Description
  Row[6]:
    CamName = Cam3P_Fp
    CamID = 6
    Description
  Row[7]:
    CamName = Cam4P
    CamID = 7
    Description
  Row[8]:
    CamName = Cam4P_Fp
    CamID = 8
    Description
  Row[9]:
    CamName = Cam5P
    CamID = 9
    Description
  Row[10]:
    CamName = Cam5P_Fp
    CamID = 10
    Description
  Row[11]:
    CamName = Cam6P
    CamID = 11
    Description
  Row[12]:
    CamName = Cam6P_Fp
    CamID = 12
    Description
```

### axCfgSpin.axis - MCP1_PLC_201/mappMotion/axCfgSpin.axis
```
Element gAxSpin (Type=axis)
  BaseTypeIsReadOnly = 0
  BaseType = RotaryPeriodic
    MeasurementUnitIsReadOnly = 0
    MeasurementUnit = 5059636
    MeasurementResolutionIsReadOnly = 0
    MeasurementResolution = 0.01
    CountDirectionIsReadOnly = 0
    CountDirection = Inverse
    PeriodSettings:
      Period = 1.0
  MovementLimitsIsReadOnly = 0
  MovementLimits = Internal
    Position:
      LowerLimitMin = -1.79769313486231E308
      UpperLimitMax = 1.79769313486231E308
      LowerLimit = -1000.0
      UpperLimit = 1000.0
    VelocityIsReadOnly = 0
    Velocity:
      VelocityMax = 3.4E38
      Velocity = 50
    AccelerationIsReadOnly = 0
    Acceleration:
      AccelerationMax = 3.4E38
      Acceleration = 25
    DecelerationIsReadOnly = 0
    Deceleration:
      DecelerationMax = 3.4E38
      Deceleration = 200
  Alarms = MpAlarmX
```

### axCfgZ.axis - MCP1_PLC_201/mappMotion/axCfgZ.axis
```
Element gAxZ (Type=axis)
  BaseTypeIsReadOnly = 0
  BaseType = LinearBounded
    MeasurementUnit = 5066068
    MeasurementResolutionIsReadOnly = 0
    MeasurementResolution = 0.001
    CountDirectionIsReadOnly = 0
    CountDirection = Inverse
  MovementLimitsIsReadOnly = 0
  MovementLimits = Internal
    Position:
      LowerLimitMin = -1.79769313486231E308
      UpperLimitMax = 1.79769313486231E308
      LowerLimit = 17
      UpperLimit = 3354
    VelocityIsReadOnly = 0
    Velocity:
      VelocityMax = 3.4E38
      Velocity = 125
    AccelerationIsReadOnly = 0
    Acceleration:
      AccelerationMax = 3.4E38
      Acceleration = 30
    DecelerationIsReadOnly = 0
    Deceleration:
      DecelerationMax = 3.4E38
      Deceleration = 250
  Alarms = MpAlarmX
```

- Safety project (password-protected, skipped)

## Configuration EchCm_P3

### vAxHwCfg.purevaxcfg - MCP1_PLC_201/mappMotion/Handwheel/vAxHwCfg.purevaxcfg
```
Element vAxHwCfg (Type=purevaxcfg)
  TypeID = PureVAxConfig
  PureVAxis:
    AxisReference = gvAxHw
    Homing:
      Mode = Direct
        Position = 0.0
        ReferencePulse = NotUsed
      RestorePositionVariable
    JerkFilter = NotUsed
    GeneralPurposeAxisInterface = Used
      MechanicalElements:
        Gearbox:
          InputIsReadOnly = 0
          Input = 1
          OutputIsReadOnly = 0
          Output = 1
        RotaryToLinearTransformation:
          ReferenceDistanceIsReadOnly = 0
          ReferenceDistance = 360
      EncoderLink = OneEncoder
        PositionEncoder = External
          LinesPerRevolution = 400
          PositionType = Incremental
          PositionSource = VariableDINT
            PVMapping = ::owsPendant.HandwheelCounter
          ValidityCheck:
            ModuleOk = Variable
              PVMapping = ::ModStat_OWS_PLK1.Slot05ModuleOk
            StaleData = NotUsed
          ReferencePulse = NotUsed
          PositionFilter:
            PositionFilterTimeConstant = 0.0
            ExtrapolationTime = 0.0
      Controller:
        ModeIsReadOnly = 0
        Mode = PositionController
          Position:
            ProportionalGain = 50.0
            IntegrationTime = 0.0
            PredictionTime = 0.01
            TotalDelayTime = 0.01
            MaximumProportionalAction = 1e30
            MaximumIntegralAction = 0.0
      StopReaction:
        Quickstop = DecelerationLimit
        DriveError = DecelerationLimit
      MovementErrorLimits:
        PositionError = 0.0
      DigitalInputs:
        HomingSwitch:
          Source = NotUsed
          Level = High
        PositiveLimitSwitch:
          Source = NotUsed
          Level = High
        NegativeLimitSwitch:
          Source = NotUsed
          Level = High
        Trigger1:
          Source = NotUsed
          Level = High
        Trigger2:
          Source = NotUsed
          Level = High
        Quickstop:
          Input = NotUsed
      StatusInputs:
        PoweredOn:
          Source = NotUsed
        CommunicationReady:
          Source = NotUsed
        ReadyForPowerOn:
          Source = NotUsed
        ErrorReactionActive:
          Source = NotUsed
        Error:
          Source = NotUsed
        ErrorID:
          Source = NotUsed
        Warning:
          Source = NotUsed
        WarningID:
          Source = NotUsed
      ControlOutputs:
        PowerOn = NotUsed
        ErrorReset = NotUsed
        BrakeControl = NotUsed
        SetSpeed = NotUsed
```

### axCfgZ.axis - MCP1_PLC_201/mappMotion/axCfgZ.axis
```
Element gAxZ (Type=axis)
  BaseTypeIsReadOnly = 0
  BaseType = LinearBounded
    MeasurementUnit = 5066068
    MeasurementResolutionIsReadOnly = 0
    MeasurementResolution = 0.001
    CountDirectionIsReadOnly = 0
    CountDirection = Standard
  MovementLimitsIsReadOnly = 0
  MovementLimits = Internal
    Position:
      LowerLimitMin = -1.79769313486231E308
      UpperLimitMax = 1.79769313486231E308
      LowerLimit = -4000
      UpperLimit = 4000.0
    VelocityIsReadOnly = 0
    Velocity:
      VelocityMax = 3.4E38
      Velocity = 10
    AccelerationIsReadOnly = 0
    Acceleration:
      AccelerationMax = 3.4E38
      Acceleration = 10
    DecelerationIsReadOnly = 0
    Deceleration:
      DecelerationMax = 3.4E38
      Deceleration = 10
  Alarms = MpAlarmX
```

## Logical view

Binary libraries used (declarations not repeated): operator, runtime, standard, brsystem, sys_lib, AsBrMath, AsBrStr, astime, AsIecCon, McBase, MpAxis, McAcpAx, McPureVAx, McAxis, MpBase, McDS402Ax, SfDomain, MpRecipe, MpAlarmX 5.17.0, CoTrace, AsZip, FileIO

### Global.typ - Global data types
```iecst
(********************************************************************
 * COPYRIGHT -- General Atomics
 ********************************************************************
 * File: Global.typ
 * Author: J. Sheeron
 ********************************************************************
 * Global data types of project 305841-E00002
 ********************************************************************)

TYPE
  (****************************************)
  (***** Depth to Angle Lookup ************)
  (****************************************)

	sXYTableReal50 : STRUCT
    numberOfVals : USINT := 0; (* number of values defined *)
		xVals : ARRAY[0..49]OF REAL;
		yVals : ARRAY[0..49]OF REAL;
	END_STRUCT;

	sXYTableLu150 : STRUCT
    T1 : sXYTableReal50;
    T2 : sXYTableReal50;
    T3 : sXYTableReal50;
	END_STRUCT;

  (****************************************)
  (***** Workpiece related structures *****)
  (****************************************)

  (***** Information about a specific part *)

  sWp_Part : STRUCT (* a specific part *)
    isZCalibrated : BOOL; (* position is calibrated to process *)
    isZIndexed : BOOL; (* set when Z is at a proper index -- position is an integer multiple of index distance *)
    isOutECalibrated : BOOL; (* position is calibrated to process *)
    isInECalibrated : BOOL; (* position is calibrated to process *)
    cutPassCount : USINT; (* which cut pass is the process on *)
    zIndexCount : USINT; (* which index is Z on -- An integer rounded version of zIndexLRCount. *)
    zIndexCountSuccess : USINT; (* last index with a successful cut *)
    zIndexLRCount : LREAL; (* which index is Z on -- should normally be an integer. An LREAL for position compatability and so a proper index can be calculated *)
    serialNumber : STRING[25]; (* Part Serial Number *)
    partDfn : sWp_PartDfn; (* Part Definition used for this part *)
  END_STRUCT;

  (***** Information about a configuration or machine setup *)
  sWp_CuttingHead :	STRUCT
    (* changes to cut profile values are detected to enable/disable cam table loading *)
    StartOfCutProfile : BOOL := FALSE;
    finishingPass : BOOL; (* finishing pass yes or no *)
    passCount : USINT; (* number of passes *)
    totalDepth : REAL; (* mm, finished depth *)
    finishingPassDepth : REAL; (* mm, finishing pass depth *)
    depthAdjAngle : LREAL; (* degrees, arc over which cut depth is adjusted. LREAL for position compatibility *)
    cutOverrunAngle : LREAL; (* degrees, arc len to overrun the last pass. LREAL for position compatibility *)
    EndOfCutProfile : BOOL := FALSE;
    feedRate : REAL; (* mm/sec, feed rate *)
    retractRate : REAL; (* deg/sec, velocity used when retracting the cutters *)
    accel : REAL;
    decel : REAL;
    setZeroOffset : REAL := 0.0; (* degrees. Offset applied when set zero is requested. *)
    depthMod : REAL := 0.0; (* mm, adjusment to the calculated finished depth *)
    offsetLimitPositive : LREAL; (* positive offset angle limit *)
    offsetLimitNegative : LREAL; (* negative offset angle limit *)

  END_STRUCT;

  sWp_Spindle :	STRUCT
    nomRpm : REAL; (* RPM, nominal *)
    accel : REAL;
    decel : REAL;
  END_STRUCT;

  sWp_ZAxis :	STRUCT
    indexSpeed : REAL; (* mm/sec *)
    accel : REAL;
    decel : REAL;
    indexDist : LREAL; (* mm. Index distance *)
    setZeroOffset : LREAL := 0.0; (* degrees. Offset applied when set zero is requested. *)
    zMod : LREAL := 0.0; (* mm, adjustment to Z position *)
    startOfCutPos : LREAL; (* position corresponding to index #1 -- start of cutting *)
    loadUnloadPos : LREAL; (* position to load/unload *)
  END_STRUCT;

  sWp_CfVfd :	STRUCT
    isInPressureControl : BOOL; (* H: Pressure ctrl, L: Speed Control *)
    runSpeedManualCtrl : REAL; (* rpm, manual run speed *)
    pressureSpAutoCtrl : REAL; (* psi, auto pressure setpoint *)
    accel : REAL;
    decel : REAL;
    eocCutoutWaitTime : TIME; (* how long to wait while idle at the end of a cycle before shutting off the cutting fluid *)
  END_STRUCT;

  sWp_PartDfn :	STRUCT  (* a part definition, but not a specific part *)
    number : STRING[15]; (* Part Number *)
    name : STRING[40]; (* Part Name *)
    nomId : REAL; (* mm, nominal inside diameter *)
    nomCutLength : LREAL; (* mm. Nominal length that cuts are made over. LREAL to be compatible with motion system *)
  END_STRUCT;

  sWp_Configuration : STRUCT
    name : STRING[40]; (* Config Name *)
    (* partDfn : sWp_PartDfn;  Part Definition *)
    startOfCfg : BOOL := FALSE;
    cuttingHead : sWp_CuttingHead;
    spindle : sWp_Spindle;
    zAxis : sWp_ZAxis;
    cfVfd : sWp_CfVfd;
    endOfCfg : BOOL := FALSE;
  END_STRUCT;

  (****************************************)
  (***** Hardware related structures  *****)
  (****************************************)

  sRioModuleHealth : STRUCT
    Slot01ModuleOk : BOOL;
    Slot02ModuleOk : BOOL;
    Slot03ModuleOk : BOOL;
    Slot04ModuleOk : BOOL;
    Slot05ModuleOk : BOOL;
    Slot06ModuleOk : BOOL;
    Slot07ModuleOk : BOOL;
    Slot08ModuleOk : BOOL;
    Slot09ModuleOk : BOOL;
    Slot10ModuleOk : BOOL;
    Slot11ModuleOk : BOOL;
    Slot12ModuleOk : BOOL;
    Slot13ModuleOk : BOOL;
    Slot14ModuleOk : BOOL;
    Slot15ModuleOk : BOOL;
    Slot16ModuleOk : BOOL;
    Slot17ModuleOk : BOOL;
    Slot18ModuleOk : BOOL;
    Slot19ModuleOk : BOOL;
    Slot20ModuleOk : BOOL;
    Slot21ModuleOk : BOOL;
    Slot22ModuleOk : BOOL;
    Slot23ModuleOk : BOOL;
    Slot24ModuleOk : BOOL;
    Slot25ModuleOk : BOOL;
    Slot26ModuleOk : BOOL;
    Slot27ModuleOk : BOOL;
    Slot28ModuleOk : BOOL;
    Slot29ModuleOk : BOOL;
    Slot30ModuleOk : BOOL;
    Slot31ModuleOk : BOOL;
    Slot32ModuleOk : BOOL;
  END_STRUCT;

END_TYPE
```

### Global.var - Global variables
```iecst
VAR CONSTANT
  INVALID_SENTINEL : DINT:= -9999;
  INVALID_SENTINEL_REAL : REAL:= -9999.0;
  INVALID_SENTINEL_LREAL : LREAL:= -9999.0;

  (* Axis count is set here rather than in PlcLogic so it can be used to define arrays *)
  AXIS_COUNT : DINT := 8;

END_VAR

VAR RETAIN

  (* Retained and here in global so they can be permanent variables *)

  (* Tables used to lookup inner eccentric offset angles given a depth,
  and lookup depth given an angle.
  50 element max, per lookup table, so break the lookup into pieces. *)
	gr_depthToAngleLu : sXYTableLu150;
	gr_angleToDepthLu : sXYTableLu150;

  (* Part and Machine cfg *)
  gr_CfgCurrent : sWp_Configuration;
  gr_PartCurrent :sWp_Part;
  gr_CfgSaved : ARRAY[0..19] OF sWp_Configuration;
  gr_PartSaved : ARRAY[0..19] OF sWp_Part;

  (* Axis restore positions *)
  gr_AxSpindleRestorePos : McAcpAxRestorePosType;
  gr_AxOutERestorePos : McAcpAxRestorePosType;
  gr_AxInERestorePos : McAcpAxRestorePosType;
  gr_AxZRestorePos : McAcpAxRestorePosType;

  (* axis travel limits *)
  (* Set here in global so this can be made permanent *)
  gr_AxisPositionLimits : ARRAY[0..AXIS_COUNT] OF sMot_PositionLimits;

  (* analog input params *)
  gr_AI_FT_CFFlow_Params : sAnalogInputParams;
  gr_AI_LT_CFTankLevel_Params : sAnalogInputParams;
  gr_AI_PT_CFPumpOutlet_Params : sAnalogInputParams;
  gr_AI_PT_CFFilterOutlet_Params : sAnalogInputParams;
  gr_AI_DP_CFFilter_Params : sAnalogInputParams; (* virtual input derrived from 2 PTs *)

  (* digital input params *)
  gr_DI_LSL_CFTank_Params : sDigitalInputParams;
  gr_DI_ZS_CFTankLocator_Params : sDigitalInputParams;
  gr_DI_JI_480VACOk_Params : sDigitalInputParams;

  (* production step TO and min values *)
  (* indexes correspond to ePROD_CYCLE_STEP values *)
  gr_ProdModeStepTOs   : ARRAY[0..40] OF TIME; (* step Timeout time values *)
  gr_ProdModeStepMins  : ARRAY[0..40] OF TIME; (* step minimum time values *)

END_VAR

VAR

END_VAR
```

### Logic.typ
```iecst
TYPE
  eAXIS_DESIGNATION :
    ( (* Physical Axes *)
    AD_UNKNOWN := 0,
    AD_SPINDLE := 1,
    AD_OUTER_ECCENTRIC := 2,
    AD_INNER_ECCENTRIC := 3,
    AD_Z := 4,
    (* Other axes *)
    AD_X := 5, (* depth *)
    AD_Y := 6, (* used ? *)
    (* virtual axis *)
    AD_HANDWHEEL := 7,
    (* VFD axis *)
    AD_CF_VFD := 8
  ) := AD_UNKNOWN;

  (* Machine specific HMI axis requests. Intended to have one of these structures per axis. *)
  sHmiAxisReqs : STRUCT
    (* Boolean requests in this section. *)
    (* (none *)
    (* numerical requests *)
    (* (none *)
    (* hmi move type and direction selection related *)
    absMoveEnable : BOOL := TRUE; (* allow move type selection by default *)
    relMoveEnable : BOOL := TRUE;
    velMoveEnable : BOOL := TRUE;
    directionPosEnable : BOOL := TRUE; (* allow direction selection by default *)
    directionNegEnable : BOOL := TRUE;
    directionShortestEnable : BOOL := TRUE;
    moveDistanceEnable : BOOL := TRUE; (* enable params by default *)
    movePositionEnable : BOOL := TRUE;
    gearInEnable : BOOL := FALSE; (* coodinated axis gear in enabled *)
    shiftEnable : BOOL := FALSE; (* coordinated axis gear offset or phase shift  enabled *)
    camInEnable : BOOL := FALSE; (* coordinated axis cam in enabled *)
    disengageEnable : BOOL := FALSE; (* coordinated axis cam in enabled *)
    moveDesignation: DINT := -1; (* per hmi. 0: Abs, 1: Rel, 2:Vel or Jog, -1 is no selection. See fctDecodeHmiMoveType *)
    direction: DINT := -1; (* per hmi. 0: pos, 1: neg, 2: shortest, -1 is no selection. See fctDecodeHmiDirection *)
    (* axis designation. Two different data types for convenience. *)
    axisNo : USINT := 0; (* default to initial so setting a value can be detected. USINT for easy use in loops *)
    axisDesignation : eAXIS_DESIGNATION := AD_UNKNOWN; (* default to initial so setting a value can be detected *)
  END_STRUCT;

  (* motion params derrived from machine/part config and process point *)
  sPartMotion : STRUCT
    camTableLoaded : BOOL := FALSE; (* True if cam table was calculated and loaded after HMI changes were made *)
    totalZIndexes : USINT; (* number of Z Indexes needed to process a part *)
    passCountCurrent : USINT; (* pass counter *)
    prodCycleStepCurrent : ePROD_CYCLE_STEP; (* last completed production cycle step *)
    nominalPassDepth : REAL; (* mm. cut pass depth *)
    currentCutterDepth : REAL; (* mm. current cutter depth *)
    nominalCutVelocity : REAL; (* deg/sec. Inner and Outer Eccentric velocity while cutting. Derived from feed rate. *)
    totalOperationDistance : LREAL; (* degrees. (number of passes * (360 + over cut angle)) + ((number of passes + 1) * cut in angle) *)
    totalPassDistance : LREAL; (* degrees. (360 + over cut angle + cut in angle *)
    startOfOperationDrivePosition : LREAL; (* degrees. Outer Ecc drive position where this operation started. LREAL to be compatible with motion positions *)
    endOfAdjAzimuth : LREAL; (* degrees. Calculated azimuth position at of adj for current pass. LREAL to be compatible with motion positions *)
    endOfPassAzimuth : LREAL; (* degrees. Calculated azimuth position at end of the pass. LREAL to be compatible with motion positions *)
    endOfOperationAzimuth : LREAL; (* degrees. Calculated azimuth position at end of the operation. LREAL to be compatible with motion positions *)
    passDistanceTraveled : LREAL; (* degrees. How far have we traveled during this pass. LREAL to be compatible with motion positions *)
    cutDistanceTraveled : LREAL; (* degrees. How far have we traveled during this cut. LREAL to be compatible with motion positions *)
  END_STRUCT;

  (* Machine specific HMI process requests. Intended to have one of these per machine or otherwise as needed, but not per axis. *)
  sHmiProcessReqs : STRUCT
    (* Boolean requests in this section. *)
    (* NOTE/CAUTION These request bits may get cleared/copied by memcpy/memclr
    So be careful about adding boolean requests outside of this section.
    See ClearManualReqs action for example, in OmSaveDev program.
    Bool requests above StartOfClearedRequests won't get auto cleared *)
    StartOfClearedRequests : BOOL := FALSE;
    reqAxesReset : BOOL := FALSE;
    cfReqRun : BOOL := FALSE;
    cfReqStop : BOOL := FALSE; (* NOTE: Stop triggers SM Halt directly. This allows stopping from the HMI even in the wrong mode *)
    zReqMoveUpLimit : BOOL := FALSE;
    zReqMoveDownLimit : BOOL := FALSE;
    zReqMoveLUnL : BOOL := FALSE;
    zReqMoveSoc : BOOL := FALSE;
    zReqMoveIndexUp : BOOL := FALSE;
    zReqMoveIndexDown : BOOL := FALSE;
    zReqPosSocUseCurrent : BOOL := FALSE; (* set SOC to use the current position *)
    zReqPosSocUseSpecified :  BOOL := FALSE; (* set SOC to use the specified position *)
    zReqPosLUnLUseCurrent : BOOL := FALSE; (* set load/unload to use the current position *)
    zReqPosLUnLUseSpecified :  BOOL := FALSE; (* set load/unload to use the specified position *)
    cuttingHeadMoveReqRetract : BOOL := FALSE;
    EndOfClearedRequests : BOOL := FALSE;
    (* NOTE/CAUTION Bool requests below EndOfClearedRequests won't get auto cleared *)
    camReqCalcTable : BOOL := FALSE; (* calculate a new cam table. *)
    calCalcTableEnable : BOOL := FALSE; (* enable hmi request PB *)
    cfIsInPressureControl : BOOL := FALSE; (* H: Pressure ctrl, L: Speed Control *)
    cfRunEnable : BOOL := FALSE; (* enable hmi request PB *)
    zMoveUpReqEnable : BOOL := FALSE; (* enable hmi request PBs *)
    zMoveDownReqEnable : BOOL := FALSE; (* enable hmi request PBs *)
    zMoveToSocReqEnable : BOOL := FALSE; (* enable hmi request PBs *)
    zMoveToLUnLReqEnable : BOOL := FALSE; (* enable hmi request PBs *)
    (* numerical values used with requests *)
    cfRpmCmd : REAL;
    cfPsiCmd : REAL;
    zReqPosSoc : LREAL;
    zReqPosLUnL : LREAL;
  END_STRUCT;

  (* cutting fluid vfd params is defined globally so multiple programs can have scope *)
  sCuttingFluidVfd : 	STRUCT
    isModuleOk : BOOL; (* H: interface is seen on the I/O network *)
    isAllowedToStart : BOOL; (* H: Allow to start *)
    isAllowedToRun : BOOL; (* H: Allow to run, L: Shutdown *)
    isLocated : BOOL; (* H: tank is located *)
    isRunning : BOOL; (* H: Drive is enabled *)
    isFlowEstablished : BOOL; (* H: Flow is detected *)
    isAlmLoFlow : BOOL; (* Lo flow shutdown *)
    isWarnLoFlow : BOOL; (* Lo flow warning *)
    isAlmLoLvlSw : BOOL; (* L: low level swtich in alarm *)
    isAlmLoFluid : BOOL; (* Lo Lo fluid level shutdown *)
    isWarnLoFluid : BOOL; (* Lo fluid level warning *)
    isAlmLoOutletPressure : BOOL; (* Lo Lo outlet pressure shutdown *)
    isWarnLoOutletPressure : BOOL; (* Lo outlet pressure warning *)
    isAlmHiOutletPressure : BOOL; (* Hi outlet pressure shutdown *)
    isWarnHiOutletPressure : BOOL; (* Hi outlet pressure warning *)
    isWarnLoFilterDp : BOOL;
    isWarnHiFilterDp : BOOL;
    isAlmSummary : BOOL; (* one of the below alarms is active *)
    isWarnSummary : BOOL; (* one of the below alarms is active *)
    StdStatus : UINT; (* DS402 standardized status *)
    DevSpecStatus : UINT; (* device specific status *)
    StdError : UINT; (* DS402 standardized error code *)
    DevSpecError : UINT; (* device specific error code *)
    VelCommanded : INT; (* speed ref rpm after ramp *)
    VelAct : INT; (* speed actual rpm *)
  END_STRUCT;

  sCyclePermissives : STRUCT
    isOmOk : BOOL; (* operating mode is okay *)
    isCfRdy : BOOL;
    isCfFlowEstablished : BOOL;
    allowCycleStart : BOOL; (* H: cycle start is allowed *)
    allowCycleRun : BOOL; (* H: Allow Run, L: Cycle Stop. Maintain high to allow cycle to run *)
  END_STRUCT;

  sOperatingMode : 	STRUCT
    (* requests *)
    ReqEmoReset : BOOL := FALSE;
    HmiReqCycleStart : BOOL := FALSE;
    HmiReqCycleStop : BOOL := FALSE;
    ReqCycleStart : BOOL := FALSE; (* pb or hmi *)
    ReqCycleStop : BOOL := FALSE; (* pb or hmi *)
    isInCycle : BOOL := FALSE; (* cycle has started and is running *)
    isInCycleHold : BOOL := FALSE; (* in cycle, but stopped at a hold point *)
    isStopping : BOOL := FALSE; (* cycle has started, but is being stopped *)
    (* cycle cfg *)
    ShutOffCfBeforeUnload : BOOL; (* turn off cutting fluid before going to unload pos *)
    SingleCycleInclZIndex : BOOL; (* include Z index at end of single cycle cut *)
    CycleZInPlace : BOOL; (* allow cycle *)
    HmiSubMode : SINT; (* hmi selections of submode *)
    (* mode request are in a word to allow masking and easy clearing *)
    ModeReqBits : WORD := 16#0; (* see OM_xxx constants for bit *)
    SecurityLevel : WORD := SL_UNKNOWN;
    OperatingMode : WORD := OM_UNKNOWN;
    SubMode       : WORD := OM_UNKNOWN; (* see OM_xxx_SM sub mode constants *)
    SeqStep : DINT; (* TODO: Make this an enum *)
  END_STRUCT;

  sPendant : 	STRUCT
    enableSwActive : BOOL; (* H:Allow motion *)
    enableSwWiringOk : BOOL; (* H:Ok *)
    pendantAllowMoves : BOOL; (* From safety controller. H:Allow moves *)
    emoAcivated : BOOL; (* From safety controller. H:Ok, L: EMO activated *)
    emoWiringOk : BOOL; (* From safety controller. H:Ok *)
    resetReqHandwheelCount : BOOL;
    pendantPowerOk : BOOL; (* 24 VDC button/LED power *)
    encoderPowerOk : BOOL; (* 5 VDC encoder power *)
    PBInputs : ARRAY[1..9] OF BOOL; (* Raw digital input states. Elements/Bits 1-9 correspond to PB 1-9 *)
    PBStates : ARRAY[1..9] OF BOOL; (* Push Button states. Conditioned with behavior. Elements/Bits 1-9 correspond to PB 1-9 *)
    PLCmds : ARRAY[1..9] OF BOOL; (* Pilot light cmds. Elements/Bits 1-9 correspond to PB 1-9 *)
    AxisSelectInputs : ARRAY[1..3] OF BOOL; (* Raw axis select switch inputs *)
    SpeedSelectInputs : ARRAY[1..3] OF BOOL; (* Raw speed select inputs *)
    AxisSelection : eAXIS_DESIGNATION;
    SpeedSelection : REAL;
    HandwheelCounter : DINT;
    Position : REAL;
    PositionSnapshot : REAL; (* used by process to capture a position *)
    GearRatioNumerator : DINT := 100; (* gear factor of the slave / measurment resolution of the slave *)
    GearRatioDenominator : DINT := 100; (* gear factor of the master / measurment resolution of the master *)
    tmrCountResetPulse : TP;
    fbPBs : ARRAY[1..9] OF fbProcPB;
  END_STRUCT;

END_TYPE
```

### Logic.var
```iecst
VAR CONSTANT
  (* Use constants to prevent accidental change *)
  (* axis number is per eAXIS_DESIGNATION *)
  (*
  AD_UNKNOWN := 0,
  AD_SPINDLE := 1,
  AD_OUTER_ECCENTRIC := 2,
  AD_INNER_ECCENTRIC := 3,
  AD_Z := 4,
  derrived axes
  AD_X := 5,
  AD_Y := 6,
  AD_HANDWHEEL := 7,
  AD_CF_VFD := 8
  *)
  (* Axis count is set in global so it can be used to define arrays *)
  (* AXIS_COUNT : DINT := 8; *)
  (* Set max axis velocity and accel/decel *)
  (* TODO Verify *)

  (* motor rated max *)
  (* AXIS_SPINDLE_MAX_VELOCITY : REAL := (6000.0 / 3.0) / 60.0; motor rated max, scaled into process velocity in rev/sec. 6000 rpm motor, 3:1 gearbox in rps *)
  (* process max *)
  AXIS_SPINDLE_MAX_VELOCITY : REAL := (300 / 60.0) * 3.0; (* process velocity in rev/sec. 300 rpm nominal cutting. 3x to allow up to 3x nominal *)
  AXIS_SPINDLE_MAX_ACCEL : REAL := AXIS_SPINDLE_MAX_VELOCITY / 2.0; (* get to max in 2 sec *)
  AXIS_SPINDLE_MAX_DECEL : REAL := AXIS_SPINDLE_MAX_VELOCITY * 4.0; (* allow faster stops *)
  AXIS_SPINDLE_MEAS_RESOLUTION : REAL := 0.01; (* Needs to match axis configuration view >> mappMotion setting for the axis *)

  (* motor rated max *)
  AXIS_OUTE_MAX_VELOCITY : REAL := (6000.0 / 25.0) * 360 / 60.0; (* motor max in deg/sec *)
  (* process max *)
  (* AXIS_OUTE_MAX_VELOCITY : REAL := (((4.7 * 25.4) / (50.0 * 3.14159)) * 360.0 / 60.0) * 4.0; (* process max in deg/sec. 4.7 in/min converted to deg/sec. 4x to allow up to 4x nominal *)
  AXIS_OUTE_MAX_ACCEL : REAL := AXIS_OUTE_MAX_VELOCITY / 1.0; (* get to max in 1 sec *)
  AXIS_OUTE_MAX_DECEL : REAL := AXIS_OUTE_MAX_ACCEL * 4.0; (* allow faster stops *)
  AXIS_OUTE_MEAS_RESOLUTION : REAL := 0.001; (* Needs to match axis configuration view >> mappMotion setting for the axis *)

  (* motor rated max *)
  AXIS_INE_MAX_VELOCITY : REAL := (6000.0 / 25.0) * 360 / 60.0; (* motor max in deg/sec *)
  (* AXIS_INE_MAX_VELOCITY : REAL := (((4.7 * 25.4) / (50.0 * 3.14159)) * 360.0 / 60.0) * 4.0;  process max in deg/sec. 4.7 in/min converted to deg/sec. 4x to allow up to 4x nominal *)
  AXIS_INE_MAX_ACCEL : REAL := AXIS_INE_MAX_VELOCITY / 1.0; (* get to max in 1 sec *)
  AXIS_INE_MAX_DECEL : REAL := AXIS_INE_MAX_ACCEL * 4.0; (* allow faster stops *)
  AXIS_INE_MEAS_RESOLUTION : REAL := 0.001; (* Needs to match axis configuration view >> mappMotion setting for the axis *)

  (* motor rated max *)
  (* AXIS_Z_MAX_VELOCITY : REAL := (3000.0 / 60.0) * 5.0; 3000 rpm motor, 5:1 lead, mm/sec *)
  (* limit due to need for mech adjustment *)
  AXIS_Z_MAX_VELOCITY : REAL := 50.0;
  AXIS_Z_MAX_ACCEL : REAL := AXIS_Z_MAX_VELOCITY / 2.0;
  AXIS_Z_MAX_DECEL : REAL := AXIS_Z_MAX_VELOCITY * 4.0; (* allow faster stops *)
  AXIS_Z_MEAS_RESOLUTION : REAL := 0.001; (* Needs to match axis configuration view >> mappMotion setting for the axis *)

  AXIS_HW_MEAS_RESOLUTION : REAL := 0.01; (* Needs to match axis configuration view >> mappMotion setting for the axis *)

  AXIS_CFVFD_MAX_VELOCITY : REAL := 1400.0 / 60.0; (* RPM to RPS *)
  AXIS_CFVFD_MAX_ACCEL : REAL := AXIS_CFVFD_MAX_VELOCITY; (* to max in 1 sec *)
  AXIS_CFVFD_MAX_DECEL : REAL := AXIS_CFVFD_MAX_VELOCITY; (* from max in 1 sec *)

  (* Operating Mode *)
  (* in increasing order of automation no motion -> manual -> production *)
  (* requests are bit packed, so pick values for easy masking *)
  (* Use constants instead of enum so word/bit operations are legal *)
  OM_UNKNOWN : WORD             := 16#00;  (* all bits clear *)
  OM_INITIAL : WORD             := 16#01;  (* bit 0 *)
  OM_SAFE_MODE : WORD           := 16#02;  (* bit 1 *)
  OM_EMO_MODE : WORD            := 16#04;  (* bit 2 *)
  OM_CHECK_MODE : WORD          := 16#08;  (* bit 3 *)
  OM_MANUAL_MODE : WORD         := 16#10;  (* bit 4 *)
  OM_PENDANT_MODE : WORD        := 16#20;  (* bit 5 *)
  OM_PRODUCTION_MODE : WORD     := 16#40;  (* bit 6 *)
  (* sub modes *)
  OM_PROD_SM_CONTINUOUS : WORD  := 16#40; (* bit 6. Run a continuous (normal) cycle *)
  OM_PROD_SM_SINGLE : WORD      := 16#41; (* bits 6, 0. Run a single cycle *)
  OM_PROD_SM_STEPPED : WORD     := 16#42; (* bits 6, 1. Run a stepped cycle *)

  (* Security Level *)
  (* values should be in increasing levels of permsision *)
  (* Anything above 1 should have some operating permission -- i.e. can leave safe mode *)
  (* chose bits to allow easy masking and combinations *)
  (* Use constants instead of enum so word/bit operations are legal *)
  SL_UNKNOWN : WORD        := 16#0;  (* all bits clear *)
  SL_GUEST : WORD          := 16#1;  (* bit 0 *)
  SL_OPERATOR : WORD       := 16#2;  (* bit 1 *)
  SL_SUPERVISOR : WORD     := 16#4;  (* bit 2 *)
  SL_ENGINEER : WORD       := 16#8;  (* bit 3 *)
  SL_SUPERUSER : WORD      := 16#10; (* bit 4 *)

  (* process tolerances *)
  TOL_DEPTH_ZERO_DEG : LREAL := 0.1; (* degrees. Values less than this are considered zero. LREAL to be comparable to positions. TODO: Need proper value *)
  TOL_ZINDEX  : LREAL := 0.2; (* Somewhat arbitrarily TODO: determine proper value *)

  (* production mode cam ID *)
  PROD_CAM_TABLE_ID : UINT := 14;

END_VAR

VAR RETAIN
  partMotion : sPartMotion; (* calculated values for processing part. Retain to preserve dynamic values *)
END_VAR

VAR
  blink025Hz : BOOL; (* 0.25 Hz blink *)
  blink050Hz : BOOL; (* 0.50 Hz blink *)
  blink100Hz : BOOL; (* 1.00 Hz blink *)

  (* IO Module Health *)
  ModStat_PLC_201 : sRioModuleHealth;
  ModStat_OWS_PLK1 : sRioModuleHealth;
  ModStat_JB1_PLK2 : sRioModuleHealth;

  (* array of axis structures *)
  axes : ARRAY[0..AXIS_COUNT] OF sMot_Axis; (* element 0 is used as a dummy axis -- an address to reference that is not an axis *)

  (* cutting fluid VFD *)
  cfVfd: sCuttingFluidVfd;

  (* global axis commands *)
  gMotionCommands : sMot_GlobalCommands; (*command structure for global command*)

  (* Operating Mode and security level *)
  operatingMode : sOperatingMode;

  (* cycle permissives *)
  cyclePermissives : sCyclePermissives;

  (* OWS Pendant *)
  owsPendant : sPendant;

  (* HMI process specific requests *)
  hmiProcessReqs : sHmiProcessReqs; (* process specific reqs *)

  (* analog inputs *)
	AI_FT_CFFlow : sAnalogInput;
	AI_LT_CFTankLevel : sAnalogInput;
	AI_PT_CFPumpOutlet : sAnalogInput;
  AI_PT_CFFilterOutlet : sAnalogInput;
  AI_DP_CFFilter : sAnalogInput;  (* virtual input derrived from 2 PTs *)

  (* digital inputs *)
	DI_LSL_CFTank : sDigitalInput;
	DI_ZS_CFTankLocator : sDigitalInput;
  DI_JI_480VACOk : sDigitalInput;
  (* digital outputs *)
  (* pb lamps *)
  DO_PB_OWSGreen : BOOL;
  DO_PB_OWSRed : BOOL;
  (* pilot lights *)
  DO_PL_OWSGreen : BOOL;
  DO_PL_OWSAmber : BOOL;
  DO_PL_OWSRed : BOOL;
  (* becon *)
  DO_PL_OWSBeconRed : BOOL;
	DO_PL_OWSBeconAmber : BOOL;
  DO_PL_OWSBeconGreen : BOOL;

END_VAR
```

### Program Logical/PlcLogic/ProcInputs (IEC)

#### ProcInputs.st
```iecst
PROGRAM _INIT

  // **** INIT Input Processing
  // Init function blocks
  // Set the reference to the input strucures,
  // set the sentinel value, and init the fb
  // Set the channel health for the sensor to OK if the module type used does not report channel health

  // ** Analog Inputs

  // ** Cutting Fluid Pump Flow Transmitter
  // NOTE: No sensor initially fitted -- here for future use
  fbAI_FT_CFFlow._InInputStruct:= ADR(AI_FT_CFFlow);
  fbAI_FT_CFFlow._InParamsStruct := ADR(gr_AI_FT_CFFlow_Params);
  fbAI_FT_CFFlow._InSentinel:= INVALID_SENTINEL_REAL;
  fbAI_FT_CFFlow(_InSetParams:= TRUE);
  fbAI_FT_CFFlow._InSetParams:= FALSE;

  // ** Cutting Fluid Tank Level Transmitter
  // NOTE: No sensor initially fitted -- here for future use
  fbAI_LT_CFTankLevel._InInputStruct:= ADR(AI_LT_CFTankLevel);
  fbAI_LT_CFTankLevel._InParamsStruct := ADR(gr_AI_LT_CFTankLevel_Params);
  fbAI_LT_CFTankLevel._InSentinel:= INVALID_SENTINEL_REAL;
  fbAI_LT_CFTankLevel(_InSetParams:= TRUE);
  fbAI_LT_CFTankLevel._InSetParams:= FALSE;

  // ** Cutting Fluid Filter Outlet Pressure Transmitter
  fbAI_PT_CFFilterOutlet._InInputStruct:= ADR(AI_PT_CFFilterOutlet);
  fbAI_PT_CFFilterOutlet._InParamsStruct := ADR(gr_AI_PT_CFFilterOutlet_Params);
  fbAI_PT_CFFilterOutlet._InSentinel:= INVALID_SENTINEL_REAL;
  fbAI_PT_CFFilterOutlet(_InSetParams:= TRUE);
  fbAI_PT_CFFilterOutlet._InSetParams:= FALSE;

  // ** Cutting Fluid Pump Outlet Pressure Transmitter
  fbAI_PT_CFPumpOutlet._InInputStruct:= ADR(AI_PT_CFPumpOutlet);
  fbAI_PT_CFPumpOutlet._InParamsStruct := ADR(gr_AI_PT_CFPumpOutlet_Params);
  fbAI_PT_CFPumpOutlet._InSentinel:= INVALID_SENTINEL_REAL;
  fbAI_PT_CFPumpOutlet(_InSetParams:= TRUE);
  fbAI_PT_CFPumpOutlet._InSetParams:= FALSE;

  // ** Cutting Fluid Pump Filter Differential Pressure Transmitter
  // Note: This is a 'virtual' instrument -- the dp across the filter is derrived
  // from the two pressure transducers. Use the Real input type -- it does not need scaling,
  // but does need alarming.
  gr_AI_DP_CFFilter_Params.RawType := GAPIO_RWST_REAL;
  fbAI_DP_CFFilter._InInputStruct:= ADR(AI_DP_CFFilter);
  fbAI_DP_CFFilter._InParamsStruct := ADR(gr_AI_DP_CFFilter_Params);
  fbAI_DP_CFFilter._InSentinel:= INVALID_SENTINEL_REAL;
  fbAI_DP_CFFilter(_InSetParams:= TRUE);
  fbAI_DP_CFFilter._InSetParams:= FALSE;

  // ** Digital Inputs
  fbDI_JI_480VACOk._InInputStruct:= ADR(DI_JI_480VACOk);
  fbDI_JI_480VACOk._InParamsStruct:= ADR(gr_DI_JI_480VACOk_Params);
  fbDI_JI_480VACOk._InSentinel:= FALSE;
  fbDI_JI_480VACOk(_InSetParams:= TRUE);
  fbDI_JI_480VACOk._InSetParams:= FALSE;

  fbDI_LSL_CFTank._InInputStruct:= ADR(DI_LSL_CFTank);
  fbDI_LSL_CFTank._InParamsStruct:= ADR(gr_DI_LSL_CFTank_Params);
  fbDI_LSL_CFTank._InSentinel:= FALSE;
  fbDI_LSL_CFTank(_InSetParams:= TRUE);
  fbDI_LSL_CFTank._InSetParams:= FALSE;

  fbDI_ZS_CFTankLocator._InInputStruct:= ADR(DI_ZS_CFTankLocator);
  fbDI_ZS_CFTankLocator._InParamsStruct:= ADR(gr_DI_ZS_CFTankLocator_Params);
  fbDI_ZS_CFTankLocator._InSentinel:= FALSE;
  fbDI_ZS_CFTankLocator(_InSetParams:= TRUE);
  fbDI_ZS_CFTankLocator._InSetParams:= FALSE;
END_PROGRAM

PROGRAM _CYCLIC

  // Set the default params on request, and then clear the request.
  // NOTE: This is not normally needed due to global
  // permanent retained status of parameters, but use for special
  // cases like first startup after major change, or to make sure
  // values are set to known, observable values.
  IF reqSetDefaultValues THEN
    SetInputParams;
    reqSetDefaultValues := FALSE;
  END_IF;

  // **** Run the analog and digital input processing
  // The input signals are generally mapped in the I/O mapping, unless there is a
  // further conditioning or logic needed.
  // Map the ModuleOk, ChannelOk, and run the fb.
  // If the channel OK is not available in the hardware I/O mapping,
  // either do it manually, or use the Module OK for the channel ok.

  // ** Analog Inputs

  AI_FT_CFFlow.ModuleOk:= ModStat_JB1_PLK2.Slot04ModuleOk;
  fbAI_FT_CFFlow();

  AI_LT_CFTankLevel.ModuleOk:= ModStat_JB1_PLK2.Slot04ModuleOk;
  fbAI_LT_CFTankLevel();

  AI_PT_CFFilterOutlet.ModuleOk:= ModStat_JB1_PLK2.Slot05ModuleOk;
  AI_PT_CFFilterOutlet.ChannelOk := AI_PT_CFFilterOutlet.ModuleOk; // TODO: Update. Need to figure out what is needed in the IO-Link case.
  fbAI_PT_CFFilterOutlet();

  AI_PT_CFPumpOutlet.ModuleOk:= ModStat_JB1_PLK2.Slot05ModuleOk;
  AI_PT_CFPumpOutlet.ChannelOk := AI_PT_CFPumpOutlet.ModuleOk; // TODO: Update. Need to figure out what is needed in the IO-Link case.
  fbAI_PT_CFPumpOutlet();

  // The 'virtual' CF Filter DP is derrived from two real PTs across the filter/
  // And the module and channel okays. Subtract the PVs to get the new signal.
  AI_DP_CFFilter.ModuleOk:= AI_PT_CFPumpOutlet.ModuleOk AND AI_PT_CFFilterOutlet.ModuleOk;
  AI_DP_CFFilter.ChannelOk := AI_PT_CFPumpOutlet.ChannelOk AND AI_PT_CFFilterOutlet.ChannelOk;
  AI_DP_CFFilter.InRawREAL := AI_PT_CFPumpOutlet.InScaled - AI_PT_CFFilterOutlet.InScaled;
  fbAI_DP_CFFilter();

  // ** Digital Inputs
  DI_JI_480VACOk.ModuleOk := ModStat_PLC_201.Slot01ModuleOk;
  DI_JI_480VACOk.ChannelOk := DI_JI_480VACOk.ModuleOk;
  fbDI_JI_480VACOk();

  DI_LSL_CFTank.ModuleOk := ModStat_JB1_PLK2.Slot02ModuleOk;
  DI_LSL_CFTank.ChannelOk := DI_LSL_CFTank.ModuleOk;
  fbDI_LSL_CFTank();

  DI_ZS_CFTankLocator.ModuleOk := ModStat_JB1_PLK2.Slot02ModuleOk;
  DI_ZS_CFTankLocator.ChannelOk := DI_ZS_CFTankLocator.ModuleOk;
  fbDI_ZS_CFTankLocator;

END_PROGRAM

PROGRAM _EXIT
	(* Insert code here *)

END_PROGRAM
```

### Program Logical/PlcLogic/Pendant (IEC)

#### Pendant.var - Local variables
```iecst
VAR RETAIN

END_VAR

VAR CONSTANT

END_VAR

VAR

  setZeroReq : BOOL := FALSE;
  homeSeqOS : BOOL := FALSE;
(*  enableInitDone : BOOL := FALSE; *)
  axisSelection : eAXIS_DESIGNATION;
(*  fbPendantInit : fbEnablePendantInit; *)
  enabledAxisFb : fbEnabledAxis;
(*  HomeAxisFb : fbHomeAbsSeq; *)

END_VAR
```

#### Pendant.st - Init, cyclic, exit code
```iecst
PROGRAM _INIT
  // Set the PB behavior. Done in init as these should't change often
  // Behavior options are:
  // GAPIO_PBBT_DISABLED    always off
  // GAPIO_PBBT_MOMENTARY   active while pressed
  // GAPIO_PBBT_OS_ON       active for one scan (rising edge of PB)
  // GAPIO_PBBT_PRESS_ON    press to turn on
  // GAPIO_PBBT_PULSE_ON    turn on for a pulse
  // GAPIO_PBBT_PRESS_OFF   press to turn off
  // GAPIO_PBBT_TOGGLE      press to toggle
  // Buttons are as follows
  // 1 (S5)  Rdy Indicator Pressed Fct TBD    Top Left
  // 2 (S6)  not assigned                     Top Mid
  // 3 (S7)  Set Zero                         Top Right
  // 4 (S8)  Axis Enable                      Mid Left
  // 5 (S9)  Axis Disable                     Mid Mid
  // 6 (S10) Brake Off                        Mid Right
  // 7 (S11) Z Set SOC                        Bot Left
  // 8 (S12) Z Set Load/Unload                Bot Mid
  // 9 (S13) Z not assigned                   Bot Right

  owsPendant.fbPBs[1]._InPBType:= GAPIO_PBBT_DISABLED; // Rdy  Press function ?. Not assigned for now.
  owsPendant.fbPBs[2]._InPBType:= GAPIO_PBBT_DISABLED; // Not assigned, no press function
  owsPendant.fbPBs[3]._InPBType:= GAPIO_PBBT_MOMENTARY;  // Set Zero
  owsPendant.fbPBs[4]._InPBType:= GAPIO_PBBT_MOMENTARY;  // Axis Enable
  owsPendant.fbPBs[5]._InPBType:= GAPIO_PBBT_MOMENTARY;  // Axis Disable
  owsPendant.fbPBs[6]._InPBType:= GAPIO_PBBT_TOGGLE;    // Manual Brake Release
  owsPendant.fbPBs[7]._InPBType:= GAPIO_PBBT_MOMENTARY ; // Z Set Start of Cut
  owsPendant.fbPBs[8]._InPBType:= GAPIO_PBBT_MOMENTARY;  // Z Set Load/Unload
  owsPendant.fbPBs[9]._InPBType:= GAPIO_PBBT_DISABLED; // Not assigned, no press function

  (* TEST CODE -- Used to test LED and button electrical *)
  (*
  owsPendant.fbPBs[1]._InPBType:= GAPIO_PBBT_MOMENTARY; // Rdy  Press function ?. Not assigned for now.
  owsPendant.fbPBs[2]._InPBType:= GAPIO_PBBT_MOMENTARY; // Not assigned, no press function
  owsPendant.fbPBs[3]._InPBType:= GAPIO_PBBT_MOMENTARY;  // Set Zero
  owsPendant.fbPBs[4]._InPBType:= GAPIO_PBBT_MOMENTARY;  // Axis Enable
  owsPendant.fbPBs[5]._InPBType:= GAPIO_PBBT_MOMENTARY;  // Axis Disable
  owsPendant.fbPBs[6]._InPBType:= GAPIO_PBBT_MOMENTARY;    // Brake Off
  owsPendant.fbPBs[7]._InPBType:= GAPIO_PBBT_MOMENTARY ; // Z Set Start of Cut
  owsPendant.fbPBs[8]._InPBType:= GAPIO_PBBT_MOMENTARY;  // Z Set Load/Unload
  owsPendant.fbPBs[9]._InPBType:= GAPIO_PBBT_MOMENTARY; // Not assigned, no press function
  *)

  // clear local home reqs and OS, and reset home fb. Set the axis to a dummy axis so
  // at least there is a reference to something
  setZeroReq := FALSE;
  // fbHomeAbs(_I_Enable := FALSE, _I_Axis := ADR(axes[AD_UNKNOWN]));

  // Init the enabled fb
  enabledAxisFb._I_PendantEnabled :=FALSE;
  enabledAxisFb._I_AxEnabled := FALSE;
  enabledAxisFb._I_AxisHandwheel := ADR(axes[AD_HANDWHEEL]);
  enabledAxisFb._I_pAxisSelected := ADR(axes[AD_UNKNOWN]); // This is dynamic, but set it to something valid
  enabledAxisFb._I_Pendant := ADR(owsPendant);
  // make sure dynamic vars (_I_pAxisSelected) are set to something when SFCInit is true
  enabledAxisFb(SFCInit:= TRUE); // inti the fb and then clear the init so it is ready to run
  enabledAxisFb.SFCInit:= FALSE;

END_PROGRAM

PROGRAM _CYCLIC

  // Allow Pendant Moves
  // No coded needed here:
  // owsPendant.pendantAllowMoves is mapped from the safety PLC: The Pendant Mode bit is sent
  // from the gray PLC to the Safe PLC. The Safe PLC sets allow moves if the wiring is okay,
  // the pendant enable button is pressed, and the mode is pendant mode.

  // Decode the axis selection
  owsPendant.AxisSelection := fctDecodeAxis(
    _InA := owsPendant.AxisSelectInputs[1],
    _InB := owsPendant.AxisSelectInputs[2],
    _InC := owsPendant.AxisSelectInputs[3],
    _InD := FALSE);

  // Decode the speed selection
  owsPendant.SpeedSelection := fctDecodeSpeed(
    _InA := owsPendant.SpeedSelectInputs[1],
    _InB := owsPendant.SpeedSelectInputs[2],
    _InC := owsPendant.SpeedSelectInputs[3],
    _InD := FALSE);

  // Call the enable axis function block. This is intended to be called all the time, and will
  // ready the machine when the pandant enable switch is pressed, and the selected axis is enabled.
  // This call assumes reference to the handwheel and pendant (both static) are set in init above.
  enabledAxisFb._I_PendantEnabled := owsPendant.pendantAllowMoves;
  enabledAxisFb._I_AxEnabled := axes[owsPendant.AxisSelection].Status.IsPoweredOn;
  enabledAxisFb._I_AxisHandwheel := ADR(axes[AD_HANDWHEEL]);
  enabledAxisFb._I_pAxisSelected := ADR(axes[owsPendant.AxisSelection]);
  enabledAxisFb._I_Pendant := ADR(owsPendant);
  enabledAxisFb();

  // Pulse count reset request
  owsPendant.tmrCountResetPulse(IN:= owsPendant.resetReqHandwheelCount, PT:= T#200ms);
  owsPendant.resetReqHandwheelCount := FALSE;

  // Process Pushbutton (PB) Inputs
  // Buttons are as follows
  // 1 (S5)  Rdy Indicator Pressed Fct TBD    Top Left
  // 2 (S6)  not assigned                     Top Mid
  // 3 (S7)  Set Zero                         Top Right
  // 4 (S8)  Axis Enable                      Mid Left
  // 5 (S9)  Axis Disable                     Mid Mid
  // 6 (S10) Brake Off                        Mid Right
  // 7 (S11) Z Set SOC                        Bot Left
  // 8 (S12) Z Set Load/Unload                Bot Mid
  // 9 (S13) not assigned                     Bot Right

  // Map the raw input into the PB FB, and run the FB.
  // Condition inputs with module OK and allow pendant moves from safety controller. This effectively
  // disables the pushbutton if pendant moves are not allowed, or the input module is not okay.
  // 1. Ready
  owsPendant.fbPBs[1](_InPBIn := owsPendant.PBInputs[1] AND ModStat_OWS_PLK1.Slot03ModuleOk AND owsPendant.pendantAllowMoves);
  owsPendant.PBStates[1] := owsPendant.fbPBs[1]._OutState;

  // 2. Not assigned
  owsPendant.fbPBs[2](_InPBIn := owsPendant.PBInputs[2] AND ModStat_OWS_PLK1.Slot03ModuleOk AND owsPendant.pendantAllowMoves);
  owsPendant.PBStates[2] := owsPendant.fbPBs[2]._OutState;

  // 3. set zero
  owsPendant.fbPBs[3](_InPBIn := owsPendant.PBInputs[3] AND ModStat_OWS_PLK1.Slot03ModuleOk AND owsPendant.pendantAllowMoves);
  owsPendant.PBStates[3] := owsPendant.fbPBs[3]._OutState;

  // 4. Axis Enable
  owsPendant.fbPBs[4](_InPBIn := owsPendant.PBInputs[4] AND ModStat_OWS_PLK1.Slot03ModuleOk AND owsPendant.pendantAllowMoves);
  owsPendant.PBStates[4] := owsPendant.fbPBs[4]._OutState;

  // 5. Axis Disable
  owsPendant.fbPBs[5](_InPBIn := owsPendant.PBInputs[5] AND ModStat_OWS_PLK1.Slot03ModuleOk AND owsPendant.pendantAllowMoves);
  owsPendant.PBStates[5] := owsPendant.fbPBs[5]._OutState;

  // 6. Brake Off
  owsPendant.fbPBs[6](_InPBIn := owsPendant.PBInputs[6] AND ModStat_OWS_PLK1.Slot03ModuleOk AND owsPendant.pendantAllowMoves);
  owsPendant.PBStates[6] := owsPendant.fbPBs[6]._OutState;

  // 7. Z Set SOC Pos
  owsPendant.fbPBs[7](_InPBIn := owsPendant.PBInputs[7] AND ModStat_OWS_PLK1.Slot04ModuleOk AND owsPendant.pendantAllowMoves);
  owsPendant.PBStates[7] := owsPendant.fbPBs[7]._OutState;

  // 8. Z Set Load/Unload Pos
  owsPendant.fbPBs[8](_InPBIn := owsPendant.PBInputs[8] AND ModStat_OWS_PLK1.Slot04ModuleOk AND owsPendant.pendantAllowMoves);
  owsPendant.PBStates[8] := owsPendant.fbPBs[8]._OutState;

  // 9. Not assigned
  owsPendant.fbPBs[9](_InPBIn := owsPendant.PBInputs[9] AND ModStat_OWS_PLK1.Slot04ModuleOk AND owsPendant.pendantAllowMoves);
  owsPendant.PBStates[9] := owsPendant.fbPBs[9]._OutState;

  (* TEST CODE. Used to test LED and button electrical. Turn on the LEDs while the buttons are pressed. *)
  (*
  owsPendant.fbPBs[1](_InPBIn := owsPendant.PBInputs[1]);
  owsPendant.PBStates[1] := owsPendant.fbPBs[1]._OutState;

  owsPendant.fbPBs[2](_InPBIn := owsPendant.PBInputs[2]);
  owsPendant.PBStates[2] := owsPendant.fbPBs[2]._OutState;

  owsPendant.fbPBs[3](_InPBIn := owsPendant.PBInputs[3]);
  owsPendant.PBStates[3] := owsPendant.fbPBs[3]._OutState;

  owsPendant.fbPBs[4](_InPBIn := owsPendant.PBInputs[4]);
  owsPendant.PBStates[4] := owsPendant.fbPBs[4]._OutState;

  owsPendant.fbPBs[5](_InPBIn := owsPendant.PBInputs[5]);
  owsPendant.PBStates[5] := owsPendant.fbPBs[5]._OutState;

  owsPendant.fbPBs[6](_InPBIn := owsPendant.PBInputs[6]);
  owsPendant.PBStates[6] := owsPendant.fbPBs[6]._OutState;

  owsPendant.fbPBs[7](_InPBIn := owsPendant.PBInputs[7]);
  owsPendant.PBStates[7] := owsPendant.fbPBs[7]._OutState;

  owsPendant.fbPBs[8](_InPBIn := owsPendant.PBInputs[8]);
  owsPendant.PBStates[8] := owsPendant.fbPBs[8]._OutState;

  owsPendant.fbPBs[9](_InPBIn := owsPendant.PBInputs[9]);
  owsPendant.PBStates[9] := owsPendant.fbPBs[9]._OutState;
 *)

  // Process Handwheel position
  // Handwheel count is mapped directly from I/O Module
  // Each A and B edge is counted, so a full AB cycle will be 4 counts
  // Take into account module and encoder power health
  // TODO: Process count into a position -- figure out algorithm
  IF owsPendant.pendantPowerOk AND owsPendant.encoderPowerOk AND ModStat_OWS_PLK1.Slot05ModuleOk AND owsPendant.pendantAllowMoves THEN
    owsPendant.Position := DINT_TO_REAL(owsPendant.HandwheelCounter) * 1.0;
  ELSE
    owsPendant.Position := 0.0;
  END_IF;

  // The PB FB up above set the PB states.
  // Now process those states -- map the pressed functions to logical functions elsewhere.
  // Use the pendant allow moves so PB button not pressed logic does not interfere with
  // logic used outside pendant mode -- brake release for example.
  IF owsPendant.pendantAllowMoves THEN
    ProcessPb1;
    ProcessPb2;
    ProcessPb3;
    ProcessPb4;
    ProcessPb5;
    ProcessPb6;
    ProcessPb7;
    ProcessPb8;
    ProcessPb9;
  END_IF;

  // Deal with set zero and home in position req and here by calling the
  // respective actions.
  // Set Zero is kicked off by PB3, and home in position is started when
  // the enable is pressed.  Both are but multi-scan operations and need
  // to continuously call the local copy of the GaMot library homing fb.
  // Wanted to keep the PB and init actions simple.
  // Use the pendant allow moves so homing logic does not interfere with
  // logic used outside pendant mode -- homing in manual mode for example.
  IF owsPendant.pendantAllowMoves THEN
    SetZeroSeq;
  ELSE
    // If not in pendant mode, make sure the home req and OS are clear
    setZeroReq := FALSE;
    homeSeqOS := FALSE;
  END_IF;

  // Process Pendant Pilot Light (PL) Outputs
  // 1. Ready Light. Illuminate on enabled and ready
  // TODO: Anything to check other than enabled?
  owsPendant.PLCmds[1] := axes[owsPendant.AxisSelection].Status.IsPoweredOn AND operatingMode.OperatingMode = OM_PENDANT_MODE;

  // 2. not assigned
  owsPendant.PLCmds[2] := FALSE;

  // 3. Set Zero -- Illuminate if axis is homed
  owsPendant.PLCmds[3] := axes[owsPendant.AxisSelection].Status.IsHomed AND operatingMode.OperatingMode = OM_PENDANT_MODE;

  // 4. Axis Enabled -- Illuminate when axis is enabled.
  owsPendant.PLCmds[4] := axes[owsPendant.AxisSelection].Status.IsPoweredOn AND operatingMode.OperatingMode = OM_PENDANT_MODE;

  // 5. Axis is Disabled -- Illuminate when axis is not enabled -- this covers the alarm state also
  owsPendant.PLCmds[5] := NOT axes[owsPendant.AxisSelection].Status.IsPoweredOn AND operatingMode.OperatingMode = OM_PENDANT_MODE;

  // 6. Brake is Off -- Illuminate if brake is off
  owsPendant.PLCmds[6] := axes[owsPendant.AxisSelection].Status.IsBrakeManuallyReleased AND operatingMode.OperatingMode = OM_PENDANT_MODE;

  // 7. Z Set SOC Pos -- Illuminate if SOC position is <> 0 and axis is homed.
  owsPendant.PLCmds[7] := gr_CfgCurrent.zAxis.startOfCutPos <> 0.0 AND axes[AD_Z].Status.IsHomed AND operatingMode.OperatingMode = OM_PENDANT_MODE;

  // 9. Z Set Load/Unload Pos -- Illuminate if load/unload position is <> 0 and axis is homed.
  owsPendant.PLCmds[8] := gr_CfgCurrent.zAxis.loadUnloadPos <> 0.0 AND axes[AD_Z].Status.IsHomed AND operatingMode.OperatingMode = OM_PENDANT_MODE;

  // 9. not assigned
  owsPendant.PLCmds[9] := FALSE;

  // TEST Code -- Test LED and button electrical. Set to button states and PB lights
  (*
  owsPendant.PLCmds[1] := owsPendant.PBStates[1];
  owsPendant.PLCmds[2] := owsPendant.PBStates[2];
  owsPendant.PLCmds[3] := owsPendant.PBStates[3];
  owsPendant.PLCmds[4] := owsPendant.PBStates[4];
  owsPendant.PLCmds[5] := owsPendant.PBStates[5];
  owsPendant.PLCmds[6] := owsPendant.PBStates[6];
  owsPendant.PLCmds[7] := owsPendant.PBStates[7];
  owsPendant.PLCmds[8] := owsPendant.PBStates[8];
  owsPendant.PLCmds[9] := owsPendant.PBStates[9];
  *)
END_PROGRAM

PROGRAM _EXIT
	(* Insert code here *)

END_PROGRAM
```

#### LocalFunctions.fun
```iecst
FUNCTION fctDecodeSpeed : REAL (* Decode 4 graycode inputs and return an axis designation *)
	VAR_INPUT
		_InA : BOOL;
		_InB : BOOL;
		_InC : BOOL;
		_InD : BOOL := FALSE;
	END_VAR
	VAR
		val : USINT := 0;
	END_VAR
END_FUNCTION

FUNCTION fctDecodeAxis : eAXIS_DESIGNATION (* Decode 4 graycode inputs and return an axis designation *)
	VAR_INPUT
		_InA : BOOL;
		_InB : BOOL;
		_InC : BOOL;
		_InD : BOOL := FALSE;
	END_VAR
	VAR
		val : USINT := 0;
	END_VAR
END_FUNCTION

FUNCTION_BLOCK fbCalcGearRatio (* Calc the handwheel:selected axis gear ratio *)
	VAR_INPUT
    _I_SlaveAxisDesignation : eAXIS_DESIGNATION;
		_I_SelectedSpeed : REAL;
	END_VAR
  VAR_OUTPUT
		_O_RatioNumerator : DINT;
		_O_RatioDenominator : DINT;
  END_VAR
	VAR
	END_VAR
END_FUNCTION_BLOCK

FUNCTION_BLOCK fbEnabledAxis
	VAR_INPUT
		SFCInit : BOOL; (*FunctionBlock initialization*)
    _I_PendantEnabled : BOOL;
    _I_AxEnabled : BOOL;
    _I_AxisHandwheel : REFERENCE TO sMot_Axis;
    _I_pAxisSelected : UDINT := 0; (* pointer to the selected axis *)
    _I_Pendant : REFERENCE TO sPendant;
	END_VAR

  VAR_OUTPUT

  END_VAR

	VAR
    axisSelected : REFERENCE TO sMot_Axis;
    currentStep : USINT := 0;
    selAxisNoPrev : DINT; (* detect changes to the selected axis *)
    selSpeedPrev : REAL; (* detect changes *)
    tmrStep : TON;
    CalcGearRatioFb : fbCalcGearRatio;
		zzInternalMemory : ARRAY[0..27] OF SINT; (*Internal memory*)
	END_VAR

  VAR CONSTANT
    STP_INIT : USINT := 0;
    STP_ENABLE_WAIT : USINT := 1;
    STP_NEW_AXIS_SEL : USINT := 2;
    STP_SETUP : USINT := 3;
    STP_ENGAGE_SEL_AX : USINT := 4;
    STP_DECOUPLE : USINT := 5;

  END_VAR
END_FUNCTION_BLOCK
```

#### fbEnabledAxis.sfc
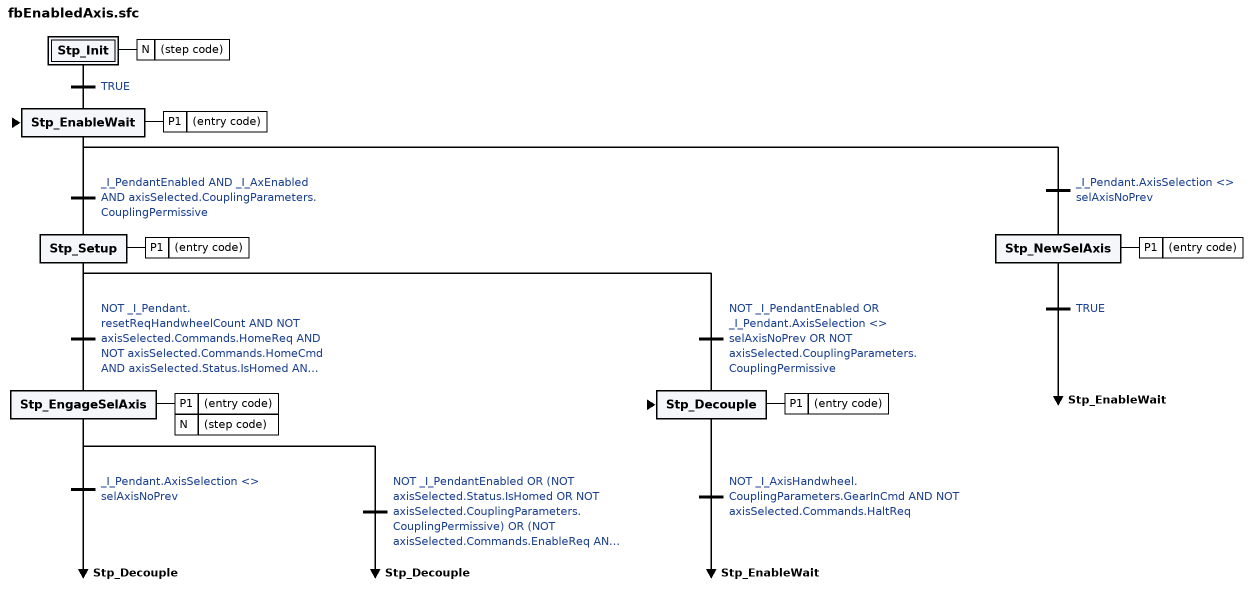
```iecst
FUNCTION_BLOCK fbEnabledAxis
INITIAL_STEP Stp_Init:
// Set current step (debugging purposes)
currentStep := STP_INIT;

// Pointers in sfc that are used in transitions
// may be dereferenced before execution begins ...
// so they need to point to something.
// Might as well pick the pointer passed in
axisSelected ACCESS _I_pAxisSelected;
END_STEP
TRANSITION FROM Stp_Init TO Stp_EnableWait:=
TRUE
END_TRANSITION
STEP Stp_EnableWait:
END_STEP
ENTRY_ACTION
// Set current step (debugging purposes)
currentStep := STP_ENABLE_WAIT;

// Get a snapshot of the axis selection so changes while processing are ignored, or at least
// handled at a time our our chosing.
// A pointer is used for access to prevent unnecessary copying of an axis structure (large)
// when 1) only a few elements are needed, and 2) the selected, and therefore referenced axis
// can change at any time.
 axisSelected ACCESS _I_pAxisSelected;

// Snapshot the selected axis number so changes can be detected
selAxisNoPrev := axisSelected.AxisNo;

// Set the virtual (handwheel) axis to use the selected axis as a slave
_I_AxisHandwheel.CouplingParameters.SlaveAxisNo := axisSelected.AxisNo;
END_ACTION
TRANSITION pendant and ax enabled FROM Stp_EnableWait TO Stp_Setup:=
// Get on with it once pendant and axis is enabled and the slave axis is okay to couple
_I_PendantEnabled AND _I_AxEnabled AND
axisSelected.CouplingParameters.CouplingPermissive
END_TRANSITION
TRANSITION new axis is selected FROM Stp_EnableWait TO Stp_NewSelAxis:=
// New axis is selected
_I_Pendant.AxisSelection <> selAxisNoPrev
END_TRANSITION
STEP Stp_NewSelAxis:
END_STEP
ENTRY_ACTION
// Set current step (debugging purposes)
currentStep := STP_NEW_AXIS_SEL;

END_ACTION
TRANSITION FROM Stp_NewSelAxis TO Stp_EnableWait:=
TRUE
END_TRANSITION
(* @SFCISJUMP := 'Stp_EnableWait' *)
STEP Stp_Setup:
END_STEP
ENTRY_ACTION
// Set current step (debugging purposes)
currentStep := STP_SETUP;

// Reset the handwheel counter. This
// guardes against rollover and allows
// starting from a predicted count.
_I_Pendant.resetReqHandwheelCount := TRUE;

// Home the virtual (handsheel) axis
// The virtual axis gets homed using direct mode
_I_AxisHandwheel.Commands.HomeReq := TRUE;
_I_AxisHandwheel.MoveParameters.HomeParams.Mode := mcHOMING_DIRECT;

// If the selected axis is not homed, request the axis be homed in position
IF NOT axisSelected.Status.IsHomed THEN
  // Set the home request for the selected axis
  axisSelected.MoveParameters.HomeParams.Mode := mcHOMING_ABSOLUTE;
  axisSelected.MoveParameters.HomeParams.Position := axisSelected.Status.Position;
  axisSelected.Commands.HomeReq := TRUE;
END_IF;
END_ACTION
TRANSITION hw counter reset and axes homed FROM Stp_Setup TO Stp_EngageSelAxis:=
// Counter reset request should be handled (low) and
// the selected axis and handwheel axis should both be homed
NOT _I_Pendant.resetReqHandwheelCount AND
NOT axisSelected.Commands.HomeReq AND
NOT axisSelected.Commands.HomeCmd AND
axisSelected.Status.IsHomed AND
NOT _I_AxisHandwheel.Commands.HomeReq AND
NOT _I_AxisHandwheel.Commands.HomeCmd AND
_I_AxisHandwheel.Status.IsHomed AND
// The axis selection should still be the same
_I_Pendant.AxisSelection = selAxisNoPrev AND
// and the slave axis coupling permissive should still be good
axisSelected.CouplingParameters.CouplingPermissive
END_TRANSITION
TRANSITION pendant disabled or new axis seleted FROM Stp_Setup TO Stp_Decouple:=
// Pendant is disabled
NOT _I_PendantEnabled OR
// New axis is selected
_I_Pendant.AxisSelection <> selAxisNoPrev OR
// slave axis coupling permissive goes away
NOT axisSelected.CouplingParameters.CouplingPermissive

END_TRANSITION
STEP Stp_Decouple:
END_STEP
ENTRY_ACTION
// Set current step (debugging purposes)
currentStep := STP_DECOUPLE;

// Clear the gear in command, and halt the slave axis
_I_AxisHandwheel.CouplingParameters.GearInCmd := FALSE;
axisSelected.Commands.HaltReq := TRUE;
END_ACTION
TRANSITION decouple and halt req FROM Stp_Decouple TO Stp_EnableWait:=
// Make sure gear in command and halt req are clear, showing they've been at least seen
NOT _I_AxisHandwheel.CouplingParameters.GearInCmd AND
NOT axisSelected.Commands.HaltReq

END_TRANSITION
(* @SFCISJUMP := 'Stp_EnableWait' *)
STEP Stp_EngageSelAxis:
// Slave (selected axis) was geared in upon entry.

// Update the gear ratio if the speed selection changes
IF _I_Pendant.SpeedSelection <> selSpeedPrev THEN
  // update the snapshot to detect future changes
  selSpeedPrev := _I_Pendant.SpeedSelection;
  // Now update the gear ratio
  CalcGearRatioFb(_I_SlaveAxisDesignation := axisSelected.AxisNo, _I_SelectedSpeed := selSpeedPrev);
  _I_Pendant.GearRatioNumerator := CalcGearRatioFb._O_RatioNumerator;
  _I_Pendant.GearRatioDenominator := CalcGearRatioFb._O_RatioDenominator;
END_IF;
END_STEP
ENTRY_ACTION
// Set current step (debugging purposes)
currentStep := STP_ENGAGE_SEL_AX;

// At this point, both the handwheel and selected
// axis should be homed, and the selected axis should be enabled.
// The handwheel does not need to be (cannot be) enabled.
// Time to engage the selected axis as a slave.

// Snapshot the speed selection so changes can be detected
selSpeedPrev := _I_Pendant.SpeedSelection;

// Set the gear ratio based on the speed and axis selected
CalcGearRatioFb(_I_SlaveAxisDesignation := axisSelected.AxisNo,_I_SelectedSpeed := selSpeedPrev);
_I_Pendant.GearRatioNumerator := CalcGearRatioFb._O_RatioNumerator;
_I_Pendant.GearRatioDenominator := CalcGearRatioFb._O_RatioDenominator;

// Gear in the slave axis as long as the permissive is met
_I_AxisHandwheel.CouplingParameters.GearInCmd := axisSelected.CouplingParameters.CouplingPermissive;
END_ACTION
TRANSITION new axis is selected FROM Stp_EngageSelAxis TO Stp_Decouple:=
// New axis is selected
_I_Pendant.AxisSelection <> selAxisNoPrev
END_TRANSITION
(* @SFCISJUMP := 'Stp_Decouple' *)
TRANSITION pendant or ax disabled FROM Stp_EngageSelAxis TO Stp_Decouple:=
// Pendant is disabled
NOT _I_PendantEnabled OR
// or the selected axis is no longer homed, or has lost coupling permissive, has lost the synchronized motion status
(NOT axisSelected.Status.IsHomed OR NOT axisSelected.CouplingParameters.CouplingPermissive) OR // OR axisSelected.Status.PlcOpenState <> mcAXIS_SYNCHRONIZED_MOTION) OR
// or selected axis is not enabled after request to do so has been processed -- this would usually be an alarm
(NOT axisSelected.Commands.EnableReq AND NOT axisSelected.Status.IsPoweredOn)
END_TRANSITION
(* @SFCISJUMP := 'Stp_Decouple' *)
END_FUNCTION_BLOCK
```
